// TwinCAT 3 PLC project STN100
// ProgramVersion: 3.1.4022.3
// libraries:
//   Tc2_Standard, * (Beckhoff Automation GmbH)
//   Tc2_System, * (Beckhoff Automation GmbH)
//   Tc3_Module, * (Beckhoff Automation GmbH)
// project tree:
//   ComLib/DUTs/General/ COM_ERROR_VALUE.TcTLEO, DEVICE_TYPE.TcTLEO
//   ComLib/DUTs/Level 2 Data link/ DEVICE_SEQUENCE.TcTLEO, INSTANCE_STATUS.TcTLEO
//   ComLib/DUTs/Level 4 Transport/ CommunicationData.TcDUT, DataGram.TcDUT, DATAGRAM_SEQUENCE.TcTLEO
//   ComLib/DUTs/Level 5 Session/ FUNCTION_TYPE.TcTLEO, INFO_FUNCTION_NUMBER.TcTLEO, SessionData.TcDUT, StatusInformationData.TcDUT
//   ComLib/DUTs/Level 6 Presentation/ ABB_ASYNC_FUNCTION_NUMBER.TcDUT, ABB_STATUS_OPERATING_MODE.TcTLEO, ABB_STATUS_RUNNING_MODE.TcTLEO, ABB_SYNC_FUNCTION_NUMBER.TcTLEO, GANTRY_ASYNC_FUNCTION_NUMBER.TcTLEO, GANTRY_STATUS.TcTLEO, PositionType.TcTLEO, StationType.TcTLEO
//   ComLib/GVL/ ComGVL.TcGVL
//   ComLib/POUs/Private/ _AllocateInstance.TcPOU, _CheckInstance.TcPOU, _DataGramSize.TcPOU, _FreeInstance.TcPOU, _GetInstance.TcPOU, _GetStatusInformation.TcPOU, _SetInstance.TcPOU, _TryOut.TcPOU (excluded from build)
//   ComLib/POUs/Public/Level 1 Physical/ NodeGetStatus.TcPOU, NodeGetType.TcPOU, NodeReadStrobe.TcPOU, NodeReadWord.TcPOU, NodeWriteStrobe.TcPOU, NodeWriteWord.TcPOU, ToAddress.TcPOU
//   ComLib/POUs/Public/Level 2 Data link/ DeviceCancel.TcPOU, DeviceClose.TcPOU, DeviceOpen.TcPOU, DeviceRead.TcPOU, DeviceStatus.TcPOU, DeviceUse.TcPOU, DeviceWrite.TcPOU
//   ComLib/POUs/Public/Level 4 Transport/ Communicator.TcPOU, DatagramCheckSum.TcPOU
//   ComLib/POUs/Public/Level 5 Session/RPC Remote Procedural Call/ ASyncProgress.TcPOU, ASyncRPC.TcPOU, RPC1.TcPOU, RPC2.TcPOU
//   ComLib/POUs/Public/Level 5 Session/Session/ SessionEnd.TcPOU, SessionInit.TcPOU, SessionSend.TcPOU
//   ComLib/POUs/Public/Level 6 Presentation/ABB/ ABBGetStatus.TcPOU
//   ComLib/POUs/Public/Level 6 Presentation/ABB/Goto/ ABBGoToConveyor1.TcPOU, ABBGoToConveyor2.TcPOU, ABBGoToHome.TcPOU, ABBGoToSensor.TcPOU, ABBGoToStorage.TcPOU, ABBGoToTable.TcPOU
//   ComLib/POUs/Public/Level 6 Presentation/ABB/IO/ ABBIORead.TcPOU, ABBIOReadValve.TcPOU, ABBIOWrite.TcPOU, ABBIOWriteValve.TcPOU
//   ComLib/POUs/Public/Level 6 Presentation/ABB/Move/ ABBMoveJAbs.TcPOU, ABBMoveJRel.TcPOU, ABBMoveLAbs.TcPOU, ABBMoveLRel.TcPOU
//   ComLib/POUs/Public/Level 6 Presentation/ABB/Pick Leave/ ABBPickLeaveConveyor1.TcPOU, ABBPickLeaveConveyor2.TcPOU, ABBPickLeaveSensor.TcPOU, ABBPickLeaveStorage.TcPOU, ABBPickLeaveTable.TcPOU, ABBProcessAssembly.TcPOU
//   ComLib/POUs/Public/Level 6 Presentation/Gantry/ GantryLeave.TcPOU, GantryPick.TcPOU, GantryStatus.TcPOU
//   ComLib/POUs/Public/Level 6 Presentation/ GetStatus.TcPOU
//   ComLib/VISUs/Object/ _VisuABBGoTo.TcVIS, _VisuABBPickLeave.TcVIS, _VisuABBStatus.TcVIS, _VisuAddressSelector.TcVIS, _VisuAddressShow.TcVIS, _VisuCommunicator.TcVIS, _VisuFunctionCall.TcVIS, _VisuGantryPickLeave.TcVIS, _VisuRPCStatusShow.TcVIS
//   ComLib/VISUs/ _TryOut.TcVIS (excluded from build)
//   / GlobalTextList.TcGTLO, PlcTask.TcTTO, Visualization Manager.TcVMO (not stored), VISU_TASK.TcTTO
//   GVLs/ GVL.TcGVL
//   POUs/ MAIN.TcPOU, PLC_PRG.TcPOU
//   VISUs/ Visualization.TcVIS
// real-time tasks:
//   TASK PlcTask: cycle T#10ms, priority 20, ADS port 350
//   TASK VISU_TASK: cycle T#100000us, priority 30, ADS port 351
// I/O:
//   DEVICE Device 1 (EtherCAT), AmsNetId 5.49.18.110.2.1
//     Term 1 (EK1200) [EK1200-5000 EtherCAT Power supply (2A E-Bus)]
//       Term 2 (EL6731) [EL6731 PROFIBUS DP Master]
//       Term 3 (EK1110) [EK1110 EtherCAT extension]
//     Term 4 (EK1100) [EK1100 EtherCAT Coupler (2A E-Bus)]
//       Term 5 (EL1008) [EL1008 8Ch. Dig. Input 24V, 3ms]
//       Term 6 (EL1008) [EL1008 8Ch. Dig. Input 24V, 3ms]
//       Term 7 (EL2008) [EL2008 8Ch. Dig. Output 24V, 0.5A]
//       Term 8 (EL2008) [EL2008 8Ch. Dig. Output 24V, 0.5A]
//       Term 9 (EK1110) [EK1110 EtherCAT extension]
//   DEVICE Device 2 (EL6731), AmsNetId 5.49.18.110.3.1
//     Box 10 (GSD Box) (Anybus-CC PROFIBUS DP-V1) // Vendor: HMS Industrial Networks Revision: 1.04
// variable links:
//   STN100/STN100 Instance <-> Device 1 (EtherCAT)/Term 4 (EK1100)/Term 6 (EL1008)
//     PlcTask Inputs/GVL.ixControlStnBit1 <-> Channel 1/Input
//     PlcTask Inputs/GVL.ixControlStnBit2 <-> Channel 2/Input
//     PlcTask Inputs/GVL.ixControlStnBit4 <-> Channel 3/Input
//     PlcTask Inputs/GVL.ixControlStnBit8 <-> Channel 4/Input
//     PlcTask Inputs/GVL.ixEmergencyStopActivated <-> Channel 8/Input
//     PlcTask Inputs/GVL.ixLightBeamAndGatesClosed <-> Channel 7/Input
//   STN100/STN100 Instance <-> Device 2 (EL6731)/Box 10 (GSD Box) (Anybus-CC PROFIBUS DP-V1)
//     PlcTask Inputs/ComGVL._iwABB <-> Module 5 (Input 1 word)/Inputs/Input 1 word_0_0
//     PlcTask Outputs/ComGVL._qwABB <-> Module 6 (Output 1 words)/Outputs/Output 1 words_1_0

CONFIGURATION STN100
    RESOURCE PLC ON TwinCAT3
        TASK PlcTask(INTERVAL := T#10ms, PRIORITY := 20);
        TASK VISU_TASK(INTERVAL := T#100000us, PRIORITY := 30);
        PROGRAM MAIN WITH PlcTask : MAIN;
        PROGRAM VisuElems_Visu_Prg WITH VISU_TASK : VisuElems.Visu_Prg;
    END_RESOURCE
END_CONFIGURATION

// ---- ComLib/DUTs/General/COM_ERROR_VALUE.TcTLEO
{library public}

(* Common error values for communication blocks *)
TYPE COM_ERROR_VALUE :
(
	COM_ERR_NOT_ENABLED:=-1,						(* En signal is false or block is not enabled *)
	COM_ERR_NO_ERROR:=0,							(* No error *)

 	(* Level 1 Errors *)
	COM_ERR_LEVEL1,									(* The physical layer failed during communication *)
	COM_ERR_LEVEL1_TIME_OUT,						(* Time out in the physical layer *)

 	(* Level 2 Errors *)
	COM_ERR_NOT_ALLOCATED,							(* Instance not allocated *)
	COM_ERR_INSTANCE,								(* Instance address (station/device) number not set or wrong *)
	COM_ERR_LEVEL2_TIME_OUT,						(* Time out in communication with device *)
	COM_ERR_LEVEL2_ERROR,							(* Error during send/receive *)
	COM_ERR_CANCEL,									(* Current operation was cancelled *)

 	(* Level 3 Errors *)
	COM_ERR_TWO_INSTANCES_OF_COMMUNICATOR,			(* Two instances of the communicator block exist in the configuration remove one *)
	COM_ERR_CHECKSUM,								(* Checksum error during datagram transfer *)

	(* Level 5 Error *)
	COM_ERR_NO_VALID_FUNCTION						(* Calls to an unknown RPC function *)
);
END_TYPE
//  COM_ERR_NOT_ENABLED = '-1'

// ---- ComLib/DUTs/General/DEVICE_TYPE.TcTLEO
{library PUBLIC}
TYPE DEVICE_TYPE :
(
	TYPE_ERROR:=-1, TYPE_SIMULATED:=0,  TYPE_ABB_1:=1, TYPE_GANTRY_1:=2
);
END_TYPE
//  TYPE_ERROR = '-1'

// ---- ComLib/DUTs/Level 2 Data link/DEVICE_SEQUENCE.TcTLEO
{library PUBLIC}
(*
Sequence for a specific device during send or receive on level 2.
This can be used for debug but is only visible inside a block.
 *)
TYPE DEVICE_SEQUENCE :
(
	DEVICE_SEQUENCE_NOP:=0,							(* No operation - free *)
	DEVICE_SEQUENCE_INIT,							(* Init of block *)
	DEVICE_SEQUENCE_WAIT_FOR_DEVICE_READY,			(* Prepare for wait and set busy to true *)
	DEVICE_SEQUENCE_WAIT_FOR_STROBE_LOW,			(* Wait until target device strobe and data are 0 *)
	DEVICE_SEQUENCE_PREPARE_SEND_RECEIVE,
	DEVICE_SEQUENCE_STROBE_HIGH,
	DEVICE_SEQUENCE_SEND_RECEIVE,					(* Transfer or read data *)
	DEVICE_SEQUENCE_ACK,
	DEVICE_SEQUENCE_WAIT_FOR_ANSWER,
	DEVICE_SEQUENCE_SET_LOW,						(* Data and strobe to 0 *)
	DEVICE_SEQUENCE_READY,							(* End of sequence will wait in this step until En=false *)

	DEVICE_SEQUENCE_TIME_OUT:=-1,					(* Tinme out during send or receive *)
	DEVICE_SEQUENCE_CANCEL:=-2,						(* An ongoing operation was canceld *)
	DEVICE_SEQUENCE_ERROR:=-3						(* An error during send/receive *)
);
END_TYPE
//  DEVICE_SEQUENCE_TIME_OUT = '-1'
//  DEVICE_SEQUENCE_CANCEL = '-2'
//  DEVICE_SEQUENCE_ERROR = '-3'

// ---- ComLib/DUTs/Level 2 Data link/INSTANCE_STATUS.TcTLEO
{library PUBLIC}
(*
 Status word for a specific device instance .
Function block DeviceUse or DeviceStatus will give you the status for a specific instance.
*)
TYPE INSTANCE_STATUS  : 
(
 	INSTANCE_STATUS_FREE:=0,							(* Instance not allocated *)
 	INSTANCE_STATUS_READY :=1,							(* Instance ready *)
 	INSTANCE_STATUS_BUSY:=2,							(* Instance is busy *)
	INSTANCE_STATUS_UNKNOWN:=3,							(* Unknown or address error *)

 	INSTANCE_STATUS_CANCEL:=-1							(* Instance cancel operation *)
);
END_TYPE
//  INSTANCE_STATUS_CANCEL = '-1'

// ---- ComLib/DUTs/Level 4 Transport/CommunicationData.TcDUT
{library PUBLIC}
(*
This is the data handler for all communications blocks.
Do not change any values inside the structure instead use existing function blocks to manipulate the data.
*)
TYPE CommunicationData :
STRUCT
	_Instance: 				BOOL := FALSE;								(*To check that we only have one instance of the communicator function block only one Instance can be true *)
	_ErrorID:				COM_ERROR_VALUE := COM_ERROR_VALUE.COM_ERR_NO_ERROR;			(* Current error value *)
	_Error:					BOOL:=FALSE	;								(* True if any error *)
	_Address:				INT:=-1;									(* Address value for device *)

	_Session:				SessionData;								(* Session data *)

	_ASyncProgress:			INT:=0;										(* Asynchronous function progress *)
	_ASyncStatus:			StatusInformationData;						(* Asynchronous function call status *)
	_ASyncStatusCounter:	UDINT:=0;									(* Counter to keep track of number of status calls *)

	_DataCounter:			UDINT:=0;									(* Datagram bytes transfered counter *)
	_DataExecute:			UDINT:=0;									(* Current datagram BYTE counter (EQ TO _DatatCounter OR <_DataCounter+SIZEOF DataGram) *)
	_Data:					DataGram;									(* Current datagram values*)
	_DataAnswer:			DataGram;									(* Datagram answer  *)

	_Status:				DATAGRAM_SEQUENCE := DATAGRAM_SEQUENCE.DATAGRAM_SEQUENCE_NOP;	(* Current status *)

	_TimeOutDevice:			TIME:=ComGvl.DEVICE_DEFAULT_TIME_OUT;				(* Device time out time *)
END_STRUCT
END_TYPE

// ---- ComLib/DUTs/Level 4 Transport/DataGram.TcDUT
{library PUBLIC}
(*
Structure to handle datagrams on level 4.
*)
TYPE DataGram :
STRUCT
	ParameterDW:		DWORD;		(* Parameter value (32 bit), purpose dependent on type of function *)
	ParameterB:			BYTE;		(* Parameter value (8 bit), purpose dependent on type of function *)

	FunctionType:		BYTE;		(* Type of function (8 bit) specifies a set of functions, the number must be based on the enumeration FUNCTION_TYPE, note that an enumeration is 16 bit and must be converted with WORD_TO_BYTE() to fit in this structure *)
	FunctionNumber: 	BYTE;		(* Specific Function (8 bit) *)

	CheckSum:			BYTE;		(* Checksum for DataGram *)
END_STRUCT
END_TYPE

// ---- ComLib/DUTs/Level 4 Transport/DATAGRAM_SEQUENCE.TcTLEO
{library PUBLIC}

(* Sequence for a specific communicator during send or receive *)
TYPE DATAGRAM_SEQUENCE : (
	DATAGRAM_SEQUENCE_ERROR:=-1,
	DATAGRAM_SEQUENCE_INIT:=-0,
	DATAGRAM_SEQUENCE_NOP,							(* No operation - free *)
	DATAGRAM_SEQUENCE_INIT_SEND,
	DATAGRAM_SEQUENCE_SEND_1,
	DATAGRAM_SEQUENCE_SEND_2,
	DATAGRAM_SEQUENCE_SEND_3,

	DATAGRAM_SEQUENCE_INIT_RECEIVE,
	DATAGRAM_SEQUENCE_RECEIVE_1,
	DATAGRAM_SEQUENCE_RECEIVE_2,
	DATAGRAM_SEQUENCE_RECEIVE_3,

	DATAGRAM_SEQUENCE_DONE
);
END_TYPE
//  DATAGRAM_SEQUENCE_ERROR = '-1'
//  DATAGRAM_SEQUENCE_INIT = '-0'

// ---- ComLib/DUTs/Level 5 Session/FUNCTION_TYPE.TcTLEO
{library PUBLIC}
(*
 Function type, to be used in DataGram structure to specify set of functions.

 Note that values <=0 are return values only.
 *)
TYPE FUNCTION_TYPE : 
(
	FUNCTION_TYPE_ERROR_BUSY:=-2,				(* Old function call is not ready  *)
	FUNCTION_TYPE_ERROR_NO_FUNCTION:=-1,		(* RPC function not found *)
	FUNCTION_TYPE_TASK_STARTED:=0,				(* ASynchronous function started *)
	FUNCTION_TYPE_ASYNC_RPC:=1,					(* ASynchronous RPC *)
	FUNCTION_TYPE_SYNC_RPC,   					(* Synchronous RPC *)
	FUNCTION_TYPE_INFORMATION					(* Synchronous RPC dedicated for status functions *)
);
END_TYPE
//  FUNCTION_TYPE_ERROR_BUSY = '-2'
//  FUNCTION_TYPE_ERROR_NO_FUNCTION = '-1'

// ---- ComLib/DUTs/Level 5 Session/INFO_FUNCTION_NUMBER.TcTLEO
{library PUBLIC}
TYPE INFO_FUNCTION_NUMBER :(
	INFO_FUNCTION_RPC_STATUS:=1,				(* Get RPC call status *)
	INFO_FUNCTION_SYSTEM_STATUS:=2				(* Get system status *)
);
END_TYPE

// ---- ComLib/DUTs/Level 5 Session/SessionData.TcDUT
{library PRIVATE}
(*
This is the session handler for all session blocks.
This structure can not be used outside of the CommunicationStructure.
Do not change any values inside the structure instead use existing function blocks to manipulate the data.
*)

TYPE SessionData :
STRUCT
	_Locked:			BOOL:=FALSE;				(* A session lock for this struct *)
	_SessionBussy:		BOOL:=FALSE;				(* If session is bussy sending data *)
	_SessionID:			INT:=0;						(* Session ID that locked this *)
	_SessionCounter:	INT:=0;						(* Sesion counter *)
END_STRUCT
END_TYPE

// ---- ComLib/DUTs/Level 5 Session/StatusInformationData.TcDUT
{library PUBLIC}
TYPE StatusInformationData :
STRUCT
	Progress:			INT:=0;					(* Progress on current RPC call 0-100 *)
	FunctionNumber:		INT:=0;					(* Curent RPC function number *)
	ReturnValue:		INT:=0;					(* Return value from previous RPC call *)
	Extra:				INT:=0;					(* Extra information *)
END_STRUCT
END_TYPE

// ---- ComLib/DUTs/Level 6 Presentation/ABB_ASYNC_FUNCTION_NUMBER.TcDUT
{library PUBLIC}
TYPE ABB_ASYNC_FUNCTION_NUMBER :(

	(* GoTo functions - No parameters *)
	ABB_ASYNC_FUNCTION_GOTO_HOME:=			11,
	ABB_ASYNC_FUNCTION_GOTO_TABLE:=			12,
	ABB_ASYNC_FUNCTION_GOTO_SENSOR:=		13,
	ABB_ASYNC_FUNCTION_GOTO_STORAGE:=		14,
	ABB_ASYNC_FUNCTION_GOTO_CONVEYOR_1:=	15,
	ABB_ASYNC_FUNCTION_GOTO_CONVEYOR_2:=	16,

	(* Pick Leav functions
	ParameterB=1 (TRUE) pick, 0 (FALSE) leave,
	ParameterW=position (if several positions exist)
	Note that Gripper is not affected by ParameterB value use separate function open or close gripper
 	*)
	ABB_ASYNC_FUNCTION_PL_TABLE:=			22,			(* Position 1=brick, 2=Rod, 3=Assembly *)
	ABB_ASYNC_FUNCTION_PL_SENSOR:=			23,
	ABB_ASYNC_FUNCTION_PL_STORAGE:=			24,  		(* Position 1-9 *)
	ABB_ASYNC_FUNCTION_PL_CONVEYOR_1:=		25,
	ABB_ASYNC_FUNCTION_PL_CONVEYOR_2:=		26,

	(* Process functions - No parameters *)
	ABB_ASYNC_FUNCTION_PROCESS_ASSEMBLY:=	32,

	(* Move functions
	Note, that xyz, rx,ry and rz must first be set by call to set functions (SYNC) *)
	ABB_ASYNC_ABS_MOVEJ_TO_POSE:=			101,
	ABB_ASYNC_ABS_MOVEL_TO_POSE:=			102,

	ABB_ASYNC_REL_MOVEJ_TO_POSE:=			111,
	ABB_ASYNC_REL_MOVEL_TO_POSE:=			112
);
END_TYPE

// ---- ComLib/DUTs/Level 6 Presentation/ABB_STATUS_OPERATING_MODE.TcTLEO
{library PUBLIC}
TYPE ABB_STATUS_OPERATING_MODE :
(
	ABB_STATUS_OPERATION_UNDEF:=0,				(* Undefined operating mode *)
	ABB_STATUS_OPERATION_AUTO:=1,				(* Automatic operating mode *)
	ABB_STATUS_OPERATION_MAN_PROG:=2, 			(* Manual operating mode MAX. 250 mm/S *)
	ABB_STATUS_OPERATION_MAN_TEST:=3 			(* Manual operating mode full speed, 100 % *)
);
END_TYPE

// ---- ComLib/DUTs/Level 6 Presentation/ABB_STATUS_RUNNING_MODE.TcTLEO

TYPE ABB_STATUS_RUNNING_MODE :
(
	ABB_STATUS_RUN_UNDEF:=0, 			(* Undefined running mode *)
	ABB_STATUS_RUN_CONT_CYCLE:=1, 		(* Continuous or cycle running mode *)
	ABB_STATUS_RUN_INSTR_FWD:=2,		(* Instruction forward running mode *)
	ABB_STATUS_RUN_INSTR_BWD:=3, 		(* Instruction backward running mode *)
	ABB_STATUS_RUN_SIM:=4, 				(* Simulated running mode *)
	ABB_STATUS_RUN_STEP_MOVE:=5 		(* MOVE instructions in forward running mode and logical instructions in continuous running mode *)
);
END_TYPE

// ---- ComLib/DUTs/Level 6 Presentation/ABB_SYNC_FUNCTION_NUMBER.TcTLEO
{library PUBLIC}
TYPE ABB_SYNC_FUNCTION_NUMBER :(
(* Set variable values
	ParameterW is the new value *)
	ABB_SYNC_FUNCTION_SET_X:=11,
	ABB_SYNC_FUNCTION_SET_Y:=12,
	ABB_SYNC_FUNCTION_SET_Z:=13,
	ABB_SYNC_FUNCTION_SET_RX:=14,
	ABB_SYNC_FUNCTION_SET_RY:=15,
	ABB_SYNC_FUNCTION_SET_RZ:=16,

(* Get variable values *)
	ABB_SYNC_FUNCTION_GET_X:=21,
	ABB_SYNC_FUNCTION_GET_Y:=22,
	ABB_SYNC_FUNCTION_GET_Z:=23,
	ABB_SYNC_FUNCTION_GET_RX:=24,
	ABB_SYNC_FUNCTION_GET_RY:=25,
	ABB_SYNC_FUNCTION_GET_RZ:=26,

(* Set pneumatic valve value
	ParameterB=1 or 0 *)
	ABB_SYNC_SET_VALVE1:=31,
	ABB_SYNC_SET_VALVE2:=32,
	ABB_SYNC_SET_VALVE3:=33,

	ABB_SYNC_GET_VALVE1:=41,
	ABB_SYNC_GET_VALVE2:=42,
	ABB_SYNC_GET_VALVE3:=43,

	ABB_SYNC_READ_DI:=101,
	ABB_SYNC_WRITE_DO:=102

);
END_TYPE

// ---- ComLib/DUTs/Level 6 Presentation/GANTRY_ASYNC_FUNCTION_NUMBER.TcTLEO
{library PUBLIC}
TYPE GANTRY_ASYNC_FUNCTION_NUMBER :(

(* GoTo functions - No parameters *)
	GANTRY_ASYNC_FUNCTION_GOTO_HOME:=		11,
	GANTRY_ASYNC_FUNCTION_GOTO_STATION:=	12,

(* Pick Leav function
	ParameterW=Station 1-4*10 + position 1-9 + Station 1-4*1000 +position 1-9 * 100
 *)
	GANTRY_ASYNC_FUNCTION_PL:=					22			(* Pick/leave at position *)
);
END_TYPE

// ---- ComLib/DUTs/Level 6 Presentation/GANTRY_STATUS.TcTLEO
{library PUBLIC}
TYPE GANTRY_STATUS :
(
	GANTRY_STATUS_NOT_ENABLED:=-1,					(* En signal is false or block is not enabled *)
	GANTRY_STATUS_NOT_READY:=0,						(* NOT ready *)
	GANTRY_STATUS_READY:=1, 							(* Auto run OK *)
	GANTRY_STATUS_INIT_MOVE:=2, 						(* Init of accelerations speeds etc *)
	GANTRY_STATUS_START_MOVE:=3,					(* Start transportation *)
	GANTRY_STATUS_MOVE_TO_STATION:=4,				(* Robot in motion *)
	GANTRY_STATUS_WAIT_CLEAR_ORDER:=5,			(* Wait until order is cleared *)
	GANTRY_STATUS_WAIT_FOR_ORDER:=6,				(* Wait for a pick or leave order *)
	GANTRY_STATUS_ORDER_ERROR:=7,				(* Error in pick or leave order *)
	GANTRY_STATUS_MOVE_TO_PICK:=8,					(* Robot picks pallet *)
	GANTRY_STATUS_WAIT_FOR_LEAVE_ORDER:=9,	(* Wait for leave order *)
	GANTRY_STATUS_ORDER_LEAVE_ERROR:=10,		(* Error in leave order *)
	GANTRY_STATUS_MOVE_TO_LEAVE:=11 				(* Robot leave pallet *)
);
END_TYPE
//  GANTRY_STATUS_NOT_ENABLED = '-1'

// ---- ComLib/DUTs/Level 6 Presentation/PositionType.TcTLEO
{library PUBLIC}
(* Position number type *)
TYPE PositionType : INT(1..9);
END_TYPE

// ---- ComLib/DUTs/Level 6 Presentation/StationType.TcTLEO
{library PUBLIC}
(* Station number type *)
TYPE StationType : INT(1..9);
END_TYPE

// ---- ComLib/GVL/ComGVL.TcGVL
{attribute 'qualified_only'}
{library PUBLIC}
VAR_GLOBAL CONSTANT
	VERSION_COM_LIBRARY:					REAL:=3.0;		(* Version number for library *)
	DEVICE_DEFAULT_TIME_OUT:		 		TIME := T#1S;	(* Default time out for single word messages to a specific device *)
END_VAR

{library private}
VAR_GLOBAL CONSTANT
	INSTANCE_MAX_NUMBER_OF_STATIONS:		INT := 6;
	INSTANCE_MAX_NUMBER_OF_DEVICES:			INT := 2;

	ADDRESS_SIMULATED:						INT := 602;
END_VAR

{library private}
VAR_GLOBAL
	
	//ProfiBusDP Communication to ABB-robot or Portal Robot (Gantry)
	{attribute 'TcSwapWord'}
	_iwABB     AT %I* : WORD;	//From ABB robot (Swaped byte order)
	_iw1Gantry AT %I* : WORD;	//From Gantry robot
	_iw2Gantry AT %I* : WORD;	
	_iw3Gantry AT %I* : WORD;	

	{attribute 'TcSwapWord'}
	_qwABB 	   AT %Q* : WORD; //To ABB robot (Swaped Byte order)
	_qw1Gantry AT %Q* : WORD; //To Gantry robot 
	_qw2Gantry AT %Q* : WORD; //To Gantry robot 
	_qw3Gantry AT %Q* : WORD; //To Gantry robot 
	
	
	




	_Instance : ARRAY  [1..INSTANCE_MAX_NUMBER_OF_STATIONS,
						   1..INSTANCE_MAX_NUMBER_OF_DEVICES]
													OF  INSTANCE_STATUS;

(*	Index 1: 1=PLC, 2="Simulated Robot",
	Index 2: 1=Strobe, 2=data  *)	
	_DataSimulatedStation:	ARRAY [1..INSTANCE_MAX_NUMBER_OF_DEVICES, 1..2] OF BYTE;


(*|                         |                                     | *)
(*|                         |                                     | *)
(*V                         V                                     V *)
(* -----------------------------------------------------------------*)


(*

(* Global Try Out variables only used by the TryOut block *)

(* Try out Communicator *)
	_miAddressNumber:			ARRAY [1..5] OF INT := [101, 201, 301, 401, 502];
	_miAddressIndex:			INT:=1;
	_fbTryOutCommunicator:		Communicator;
	_msTryOutData: 				CommunicationData;
	_mxTryOutEnable:			BOOL;

	_glAddressNameTable: 		ARRAY [1..5] OF STRING:= ['Station 100' , 'Station 200', 'Station 300', 'Station 400',  'Station 500'];
	_glAddressSelectionIndex: 	INT:=1;

	_glErrorTable:				ARRAY [ -1 .. 10] OF STRING :=
	 	['En signal is false or block is not enabled',
		 'No error',
		 'The physical layer failed during communication',
		 'Time out in the physical layer',
		 'Instance not allocated',
		 'Instance address (station/device) number not set or wrong',
		 'Time out in communication with device',
		 'Error during send/receive',
		 'Current operation was cancelled',
		 'Two instances of the communicator block exist in the configuration remove one',
		 'Checksum error during datagram transfer',
		 'Calls to an unknown RPC function'];

	_fbTryOutGetStatus:					GetStatus;
	_fbTryOutGetStatusRunning:			BOOL;
	_fbTryOutGetStatusProgress:			INT;
	_fbTryOutGetStatusProgramNumber:	INT;
	_fbTryOutGetStatusHeartBeat:		BOOL;
	_fbTryOutGetStatusError: 			BOOL;

(* ABB Functions *)
	_fbTryOutShowABB:					BOOL;

	_fbTryOutDone:						BOOL;
	_fbTryOutExecuting:					BOOL;
	_fbTryOutWaiting:					BOOL;
	_fbTryOutError:						BOOL;
	_fbTryOutProgress:					INT;

	_fbTryOutABBGetStatus:				ABBGetStatus;
	_fbTryOutABBRunMode:				ABB_STATUS_RUNNING_MODE;
	_fbTryOutABBOpMode:					ABB_STATUS_OPERATING_MODE;

	_gABBRunTable:						ARRAY [1 .. 6] OF STRING :=
		['Undefined running mode',
		'Continuous or cycle running mode',
		'Instruction forward running mode',
		'Instruction backward running mode',
		'Simulated running mode',
		'MOVE instr. in forward running and logical instr. in continuous running mode'];

	_gABBOpTable:						ARRAY [ 1 .. 4] OF STRING :=
		['Undefined operating mode',
		'Automatic operating mode',
		'Manual operating mode MAX. 250 mm/S',
		'Manual operating mode full speed, 100 %'];

	_fbTryOutABBGoToHome:				ABBGoToHome;
	_fbTryOutABBGoToHomeEn:				BOOL;

	_fbTryOutABBGoToSensor:				ABBGoToSensor;
	_fbTryOutABBGoToSensorEn:			BOOL;

	_fbTryOutABBGoToStorage:			ABBGoToStorage;
	_fbTryOutABBGoToStorageEn:			BOOL;

	_fbTryOutABBGoToTable:				ABBGoToTable;
	_fbTryOutABBGoToTableEn:			BOOL;

	_fbTryOutABBGoToConveyor1:			ABBGoToConveyor1;
	_fbTryOutABBGoToConveyor1En:		BOOL;

	_fbTryOutABBGoToConveyor2:			ABBGoToConveyor2;
	_fbTryOutABBGoToConveyor2En:		BOOL;

	_fbTryOutABBPickLeaveSensor:		ABBPickLeaveSensor;
	_fbTryOutABBPickLeaveSensorEn:		BOOL;
	_fbTryOutABBPSensor:				BOOL;

	_fbTryOutABBPickLeaveStorage:		ABBPickLeaveStorage;
	_fbTryOutABBPickLeaveStorageEn:		BOOL;
	_fbTryOutABBPStorage:				BOOL;
	_fbTryOutABBPStoragePos:			INT:=1;

	_fbTryOutABBPickLeaveTable:			ABBPickLeaveTable;
	_fbTryOutABBPickLeaveTableEn:		BOOL;
	_fbTryOutABBPTable:					BOOL;
	_fbTryOutABBPTablePos:				INT:=1;

	_fbTryOutABBPickLeaveConveyor1:		ABBPickLeaveConveyor1;
	_fbTryOutABBPickLeaveConveyor1En:	BOOL;
	_fbTryOutABBPConveyor1:				BOOL;

	_fbTryOutABBPickLeaveConveyor2:		ABBPickLeaveConveyor2;
	_fbTryOutABBPickLeaveConveyor2En:	BOOL;
	_fbTryOutABBPConveyor2:				BOOL;

(* Gantry Functions *)
	_fbTryOutShowGantry:			BOOL;

	_fbTryOutGantryPick:			GantryPick;
	_fbTryOutGantryPickEn:			BOOL;
	_fbTryOutGantryPickStation:		INT:=1;
	_fbTryOutGantryPickPos:			INT:=1;

	_fbTryOutGantryLeave:			GantryLeave;
	_fbTryOutGantryLeaveEn:			BOOL;
	_fbTryOutGantryLeaveStation:	INT:=1;
	_fbTryOutGantryLeavePos:		INT:=2;
*)
END_VAR

// ---- GVLs/GVL.TcGVL
{attribute 'qualified_only'}
VAR_GLOBAL
	

	//OPC-UA Communication to STN500 (the crane)
	{attribute 'OPC.UA.DA' := '1'}
	iToSTN500FromSTN100 : ARRAY[1..8] OF INT; (* To STN500 *)

	{attribute 'OPC.UA.DA' := '1'}
	iFromSTN500ToSTN100 : ARRAY[1..8] OF INT; (* From STN500 *)

	
	//Inputs from the sensors in controlstation
	ixControlStnBit1 AT %I* : BOOL;	
	ixControlStnBit2 AT %I* : BOOL;
	ixControlStnBit4 AT %I* : BOOL;
	ixControlStnBit8 AT %I* : BOOL;
	
	

	
	(* Gates and emergency stop, status signal *)
	ixLightBeamAndGatesClosed 	AT %I* : BOOL;
	ixEmergencyStopActivated 	AT %I* : BOOL;
	
	
	(* Light staple *)
	qxLampRed 		AT %Q*: BOOL;
	qxLampYellow 	AT %Q*: BOOL;
	qxLampGreen 	AT %Q*: BOOL;
	
	
	
END_VAR

// ---- POUs/MAIN.TcPOU
PROGRAM MAIN
VAR

END_VAR

PLC_PRG();

END_PROGRAM

// ---- POUs/PLC_PRG.TcPOU
PROGRAM PLC_PRG
VAR
	//Visualisation buttons	
	mxButtonReset	: BOOL;	
	mxButtonStart: BOOL;

	//Internal use
	mxStart: BOOL;
	mxDone: BOOL;
	mxComBusy: BOOL;
	CommData: CommunicationData;	
	
	//Motion Function Blocks
	fbCommunicator: Communicator;
	fbABBGoToHome_1: ABBGoToHome;
	fbABBGoToTable_1: ABBGoToTable;
END_VAR

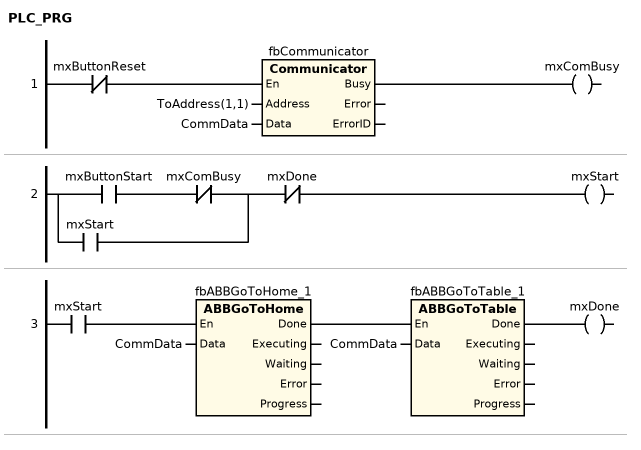
// NETWORK 1
fbCommunicator(En := NOT mxButtonReset, Address := ToAddress(1,1), Data := CommData); // Communicator
mxComBusy := fbCommunicator.Busy;

// NETWORK 2
mxStart := (mxButtonStart AND NOT mxComBusy OR mxStart) AND NOT mxDone;

// NETWORK 3
fbABBGoToHome_1(En := mxStart, Data := CommData); // ABBGoToHome
fbABBGoToTable_1(En := fbABBGoToHome_1.Done, Data := CommData); // ABBGoToTable
mxDone := fbABBGoToTable_1.Done;

END_PROGRAM

// ---- ComLib/POUs/Public/Level 4 Transport/Communicator.TcPOU
{library PUBLIC}
(* Communication interface on level 4 to be used as a single access point to communicate with external equipment (device).
    Note, that you must make one and only one instance per address (device) of this block. This block instance 
    coordinates all communication actions from all POUs to a specific device.

   The Data input must be connected to a common variable of the type CommunicationData. 
   The Data variable must then be used together with all function blocks that want to communicate with
   the specified equipment. It is possible to use function blocks on level 4-6 together with the communicator.
  However, note that it is not possible to utilize function blocks on level 1-3 together with the communicator.
*)
FUNCTION_BLOCK Communicator
VAR_INPUT
	En: 				BOOL:=TRUE;						(* Enable signal must be true during communication, set to false (pulse) to reset error and restart the block.  *)
	Address :			INT:=-1;						(* Address is the station number + device number, e.g.  202, 301, 404 and must be constant during run you can use ToAddress() function to calculate an address. *)
END_VAR
VAR_OUTPUT
	Busy: 				BOOL:=FALSE;					(* Busy is true if the block is communicating with target, otherwise false. *)
	Error: 				BOOL:=FALSE;					(* True if any error, to reset error set En to low and then back to high*)
	ErrorID: 			COM_ERROR_VALUE:=COM_ERROR_VALUE.COM_ERR_NO_ERROR;	(* The error number, if no error the output is equal to COM_ERR_NO_ERROR i.e., 0 *)
END_VAR
VAR_IN_OUT
	Data:				 CommunicationData;				(* Common data structure to connect all communication blocks that want to access this block *)
END_VAR
{library private}
VAR
	AllowToRun:		BOOL:=FALSE	;						(* If we are alone then we are allow to execute the communication*)
	Instance:		INT:=-1;							(* Device instance number *)
	DeviceType:		DEVICE_TYPE:=DEVICE_TYPE.TYPE_ERROR;
	InstanceStatus: INSTANCE_STATUS;
	Sequence: 		DATAGRAM_SEQUENCE:=DATAGRAM_SEQUENCE.DATAGRAM_SEQUENCE_INIT;
	ENWrite: 		BOOL:=FALSE;
	ENRead: 		BOOL:=FALSE;

	DataPointer:	POINTER TO BYTE;
	DataWord: 		WORD;
	StationNumber:	WORD;
	PositionNumber:	WORD;

	fbDeviceWrite: 	DeviceWrite;
	fbDeviceRead: 	DeviceRead;
	fbDeviceCancel: DeviceCancel;

	fbTON_TimeOut:	TON;							(* Only used for special sequence of gantry *)
	DEVICE_DEFAULT_TIME_OUT: INT;

	(* Variables used to change byte order in Data.ParameterDW *)
	DataHi1: BYTE; //Answer from ABB robot
	DataLo1: BYTE;
	DataHi2: BYTE;
	DataLo2: BYTE;
	DataSLo1: BYTE; //Send to ABB robot
	DataSHi1: BYTE;
	DataSHi2: BYTE;
	DataSLo2: BYTE;
END_VAR

IF NOT AllowToRun AND Instance=-1 AND En THEN
	InstanceStatus:=_GetInstance(Address);
	Instance:=0;
	Data._Address:=Address;

	IF InstanceStatus=INSTANCE_STATUS.INSTANCE_STATUS_FREE THEN
		IF DeviceOpen(Address) THEN
			Instance:=Address;
			DeviceType:=NodeGetType(Address);
			AllowToRun:=TRUE;
			Data._Instance:=TRUE;
			Error:=FALSE;
			ErrorID:=COM_ERROR_VALUE.COM_ERR_NO_ERROR;
		END_IF;
	ELSE
		Error:=TRUE;
		CASE InstanceStatus OF
			INSTANCE_STATUS.INSTANCE_STATUS_READY,  INSTANCE_STATUS.INSTANCE_STATUS_BUSY,  INSTANCE_STATUS.INSTANCE_STATUS_CANCEL:
					ErrorID:=COM_ERROR_VALUE.COM_ERR_TWO_INSTANCES_OF_COMMUNICATOR;

			INSTANCE_STATUS.INSTANCE_STATUS_UNKNOWN:
				ErrorID:=COM_ERROR_VALUE.COM_ERR_INSTANCE;
		END_CASE;
	END_IF;
END_IF;

IF AllowToRun THEN
	IF Address<>Data._Address THEN
		Busy:=FALSE;
		Error:=TRUE;
		ErrorID:=COM_ERROR_VALUE.COM_ERR_INSTANCE;
		RETURN;
	END_IF;

	fbDeviceWrite(En:=ENWrite AND En, Instance:=Instance, Data:=DataWord, TimeOut:=Data._TimeOutDevice);
	fbDeviceRead(En:=ENRead AND En, Instance:=Instance, TimeOut:=Data._TimeOutDevice);

	IF fbDeviceWrite.Error AND fbDeviceWrite.ErrorID<>COM_ERROR_VALUE.COM_ERR_CANCEL THEN
		Sequence:=DATAGRAM_SEQUENCE.DATAGRAM_SEQUENCE_ERROR;
		Error:=TRUE;
		ErrorID:=fbDeviceWrite.ErrorID;
	END_IF;

	IF fbDeviceRead.Error AND fbDeviceRead.ErrorID<>COM_ERROR_VALUE.COM_ERR_CANCEL THEN
		Sequence:=DATAGRAM_SEQUENCE.DATAGRAM_SEQUENCE_ERROR;
		Error:=TRUE;
		ErrorID:=fbDeviceRead.ErrorID;
	END_IF;

	IF En THEN
		IF DeviceType=DEVICE_TYPE.TYPE_ABB_1 THEN
			_SequenceABB_1();
		ELSIF DeviceType=DEVICE_TYPE.TYPE_GANTRY_1 THEN
			_SequenceGantry_1();
		ELSE
			Error:=TRUE;
			ErrorID:=COM_ERROR_VALUE.COM_ERR_INSTANCE;
		END_IF;
	ELSE (* En *)
		Sequence:=DATAGRAM_SEQUENCE.DATAGRAM_SEQUENCE_INIT;
		ENWrite:=FALSE;
		ENRead:=FALSE;
		Busy:=FALSE;
		Error:=FALSE;
		ErrorID:=COM_ERROR_VALUE.COM_ERR_NOT_ENABLED;

		Data._DataCounter:=0;
		Data._DataExecute:=0;
	END_IF (* En *)
END_IF;


(* Copy error to struct *)
Data._ErrorID:=ErrorID;
Data._Error:=Error;
Data._Status:=Sequence;

ACTION _SequenceABB_1:
CASE Sequence OF
			DATAGRAM_SEQUENCE.DATAGRAM_SEQUENCE_ERROR:
				Error:=TRUE;

			DATAGRAM_SEQUENCE.DATAGRAM_SEQUENCE_INIT:
				ErrorID:=COM_ERROR_VALUE.COM_ERR_NO_ERROR;
				fbDeviceCancel(En:=TRUE, Instance:=Instance);

				IF fbDeviceCancel.Done THEN
					(* Cancel set ok *)
					fbDeviceCancel(En:=FALSE, Instance:=Instance);

					(* Force DeviceWrite to execute cancel *)
					fbDeviceWrite(En:=TRUE, Instance:=Instance, Data:=DataWord, TimeOut:=Data._TimeOutDevice);
					Sequence:=DATAGRAM_SEQUENCE.DATAGRAM_SEQUENCE_NOP;
				END_IF;

			DATAGRAM_SEQUENCE.DATAGRAM_SEQUENCE_NOP:		(* Wait for order *)
				IF Data._DataCounter<>Data._DataExecute THEN
					Busy:=TRUE;
					Sequence:=DATAGRAM_SEQUENCE.DATAGRAM_SEQUENCE_INIT_SEND;
				END_IF;

			DATAGRAM_SEQUENCE.DATAGRAM_SEQUENCE_INIT_SEND:
				Data._Data.CheckSum:=DatagramCheckSum(Data._Data);
				DataPointer:= ADR(Data._Data);
				Sequence:=DATAGRAM_SEQUENCE.DATAGRAM_SEQUENCE_SEND_1;

				(* Change byte order for Intel CPU *)
				DataSLo2 := DWORD_TO_BYTE( Data._Data.ParameterDW AND 16#FF);
				DataSHi2 := DWORD_TO_BYTE( SHR(Data._Data.ParameterDW AND 16#FF00,8));
                DataSLo1 := DWORD_TO_BYTE( SHR(Data._Data.ParameterDW AND 16#FF000,16)); 
				DataSHi1 := DWORD_TO_BYTE( SHR(Data._Data.ParameterDW AND 16#FF000000,24));
				
				Data._Data.ParameterDW := BYTE_TO_DWORD( DataSHi1) OR SHL( BYTE_TO_DWORD( DataSLo1),8) OR 
                                                 SHL(BYTE_TO_DWORD( DataSHi2),16) OR SHL(BYTE_TO_DWORD( DataSLo2),24);
				
			DATAGRAM_SEQUENCE.DATAGRAM_SEQUENCE_SEND_1:
				DataWord:=BYTE_TO_WORD(DataPointer^);
				ENWrite:=TRUE;
				Sequence:=DATAGRAM_SEQUENCE.DATAGRAM_SEQUENCE_SEND_2;

			DATAGRAM_SEQUENCE.DATAGRAM_SEQUENCE_SEND_2:
				IF fbDeviceWrite.Done THEN
					ENWrite:=FALSE;
					Sequence:=DATAGRAM_SEQUENCE.DATAGRAM_SEQUENCE_SEND_3;
				END_IF;

			DATAGRAM_SEQUENCE.DATAGRAM_SEQUENCE_SEND_3:
				Data._DataCounter:=Data._DataCounter+1;
				DataPointer:=DataPointer+1;

				IF Data._DataCounter=Data._DataExecute THEN
					Sequence:=DATAGRAM_SEQUENCE.DATAGRAM_SEQUENCE_INIT_RECEIVE;
				ELSE
					Sequence:=DATAGRAM_SEQUENCE.DATAGRAM_SEQUENCE_SEND_1;
				END_IF;

			DATAGRAM_SEQUENCE.DATAGRAM_SEQUENCE_INIT_RECEIVE:
				DataPointer:= ADR(Data._DataAnswer);
				Data._DataExecute:=Data._DataExecute + INT_TO_UDINT( _DataGramSize());
				Sequence:=DATAGRAM_SEQUENCE.DATAGRAM_SEQUENCE_RECEIVE_1;

			DATAGRAM_SEQUENCE.DATAGRAM_SEQUENCE_RECEIVE_1:
				ENRead:=TRUE;
				Sequence:=DATAGRAM_SEQUENCE.DATAGRAM_SEQUENCE_RECEIVE_2;

			DATAGRAM_SEQUENCE.DATAGRAM_SEQUENCE_RECEIVE_2:
				IF fbDeviceRead.Done THEN
					ENRead:=FALSE;
					DataPointer^:=WORD_TO_BYTE(fbDeviceRead.Data);
					Sequence:=DATAGRAM_SEQUENCE.DATAGRAM_SEQUENCE_RECEIVE_3;
				END_IF;

			DATAGRAM_SEQUENCE.DATAGRAM_SEQUENCE_RECEIVE_3:
				Data._DataCounter:=Data._DataCounter+1;
				DataPointer:=DataPointer+1;

				IF Data._DataCounter=Data._DataExecute THEN
					Sequence:=DATAGRAM_SEQUENCE.DATAGRAM_SEQUENCE_DONE;
				ELSE
					Sequence:=DATAGRAM_SEQUENCE.DATAGRAM_SEQUENCE_RECEIVE_1;
				END_IF;

			DATAGRAM_SEQUENCE.DATAGRAM_SEQUENCE_DONE:
				Busy:=FALSE;

				(* Change byte order for Intel CPU *)
				DataLo1 := DWORD_TO_BYTE( Data._DataAnswer.ParameterDW AND 16#FF);
				DataHi1 := DWORD_TO_BYTE( SHR(Data._DataAnswer.ParameterDW AND 16#FF00,8));
                DataLo2 := DWORD_TO_BYTE( SHR(Data._DataAnswer.ParameterDW AND 16#FF000,16)); 
				DataHi2 := DWORD_TO_BYTE( SHR(Data._DataAnswer.ParameterDW AND 16#FF000000,24));
				
				Data._DataAnswer.ParameterDW := BYTE_TO_DWORD( DataHi1) OR SHL( BYTE_TO_DWORD( DataLo1),8) OR 
                                                SHL(BYTE_TO_DWORD( DataHi2),16) OR SHL(BYTE_TO_DWORD( DataLo2),24);
				
				IF Data._DataAnswer.CheckSum = DatagramCheckSum(Data._DataAnswer) THEN
					Data._Session._SessionCounter:=Data._Session._SessionCounter+1;
					Sequence:=DATAGRAM_SEQUENCE.DATAGRAM_SEQUENCE_NOP;
				ELSE
					ErrorID:= DINT_TO_INT( INT_TO_DINT( DATAGRAM_SEQUENCE.DATAGRAM_SEQUENCE_DONE));
					Error:=TRUE;
					Sequence:=DATAGRAM_SEQUENCE.DATAGRAM_SEQUENCE_DONE;
				END_IF;

		END_CASE;
END_ACTION

ACTION _SequenceGantry_1:
(* Note that the implementation for the Gantry does not use level 2 as intended
   it uses a mix of level 1 and 2 due to an older communication protocol in the UHS *)

		CASE Sequence OF
			DATAGRAM_SEQUENCE.DATAGRAM_SEQUENCE_ERROR:
				Error:=TRUE;
				NodeWriteWord(Address:=Instance, Channel:=0, Data:=0);									(* Write no order to pick position to crane *)
				NodeWriteWord(Address:=Instance, Channel:=1, Data:=0);									(* Write no order to pick position to crane *)

			DATAGRAM_SEQUENCE.DATAGRAM_SEQUENCE_INIT:
				ErrorID:=COM_ERROR_VALUE.COM_ERR_NO_ERROR;
				fbDeviceCancel(En:=TRUE, Instance:=Instance);

				IF fbDeviceCancel.Done THEN
					(* Cancel set ok *)
					fbDeviceCancel(En:=FALSE, Instance:=Instance);

					(* Force DeviceWrite to execute cancel *)
					fbDeviceWrite(En:=TRUE, Instance:=Instance, Data:=DataWord, TimeOut:=Data._TimeOutDevice);
					Sequence:=DATAGRAM_SEQUENCE.DATAGRAM_SEQUENCE_NOP;
				END_IF;

			DATAGRAM_SEQUENCE.DATAGRAM_SEQUENCE_NOP:		(* Wait for order *)
				IF Data._DataCounter<>Data._DataExecute THEN
					Busy:=TRUE;
					Sequence:=DATAGRAM_SEQUENCE.DATAGRAM_SEQUENCE_INIT_SEND;
				END_IF;

			DATAGRAM_SEQUENCE.DATAGRAM_SEQUENCE_INIT_SEND:
				IF Data._Data.FunctionType=FUNCTION_TYPE.FUNCTION_TYPE_INFORMATION AND Data._Data.FunctionNumber=INFO_FUNCTION_NUMBER.INFO_FUNCTION_RPC_STATUS THEN
					IF NodeReadWord(Address:=Instance, Channel:=0) =0 AND NodeReadWord(Address:=Instance, Channel:=1) =0 THEN
						Data._DataAnswer.ParameterDW:=0;
					ELSE
						Data._DataAnswer.ParameterDW:=1;
					END_IF;

					Sequence:=DATAGRAM_SEQUENCE.DATAGRAM_SEQUENCE_DONE;

				ELSIF Data._Data.FunctionType=FUNCTION_TYPE.FUNCTION_TYPE_ASYNC_RPC AND Data._Data.FunctionNumber=GANTRY_ASYNC_FUNCTION_NUMBER.GANTRY_ASYNC_FUNCTION_PL THEN
					Sequence:=DATAGRAM_SEQUENCE.DATAGRAM_SEQUENCE_SEND_1;
				ELSE
					ErrorID:=COM_ERROR_VALUE.COM_ERR_NO_VALID_FUNCTION;
					Error:=TRUE;
					Sequence:=DATAGRAM_SEQUENCE.DATAGRAM_SEQUENCE_ERROR;
				END_IF;

			DATAGRAM_SEQUENCE.DATAGRAM_SEQUENCE_SEND_1:
				(* Get pick order from Data.ParameterDW and send to gantry *)
				StationNumber:=DWORD_TO_WORD(Data._Data.ParameterDW/1000)*10;					(* 10-40 or 0*)

				IF StationNumber<>0 THEN
					PositionNumber:=DWORD_TO_WORD(Data._Data.ParameterDW/100)-StationNumber-1;	(* 0-8 *)
					PositionNumber:= ((PositionNumber/3)+1)*10 + (PositionNumber MOD 3)+1 ;				(* 11, 12, 13, 21, 22, 23, 31, 32, 33 *)

					DataWord:=Stationnumber*10+ PositionNumber;
					NodeWriteWord(Address:=Instance, Channel:=0, Data:=DataWord);							(* Write pick position to crane *)
					fbTON_TimeOut(IN:=FALSE);
					Sequence:=DATAGRAM_SEQUENCE.DATAGRAM_SEQUENCE_SEND_2;
				ELSE
					Sequence:=DATAGRAM_SEQUENCE.DATAGRAM_SEQUENCE_SEND_3;
				END_IF;

			DATAGRAM_SEQUENCE.DATAGRAM_SEQUENCE_SEND_2:
				(* Wait for ack of order *)
				fbTON_TimeOut(IN:=TRUE, PT:=ComGVL.DEVICE_DEFAULT_TIME_OUT);

				IF DataWord=NodeReadWord(Address:=Instance, Channel:=0) THEN
					Sequence:=DATAGRAM_SEQUENCE.DATAGRAM_SEQUENCE_SEND_3;
				ELSIF fbTON_TimeOut.Q THEN
					ErrorID:=COM_ERROR_VALUE.COM_ERR_LEVEL2_TIME_OUT;
					Sequence:=DATAGRAM_SEQUENCE.DATAGRAM_SEQUENCE_ERROR;
				END_IF;

			DATAGRAM_SEQUENCE.DATAGRAM_SEQUENCE_SEND_3:
				NodeWriteWord(Address:=Instance, Channel:=0, Data:=0);									(* Write no order to pick position to crane *)
				Sequence:=DATAGRAM_SEQUENCE.DATAGRAM_SEQUENCE_INIT_RECEIVE;

			DATAGRAM_SEQUENCE.DATAGRAM_SEQUENCE_INIT_RECEIVE:
				(* Get leave order from Data.ParameterDW*)
				StationNumber:=DWORD_TO_WORD(Data._Data.ParameterDW)-DWORD_TO_WORD(Data._Data.ParameterDW/100)*100;	(* 11-49 or 0*)

				IF StationNumber<>0 THEN
					PositionNumber:=StationNumber-(StationNumber/10)*10-1;									(* 0-8 *)
					PositionNumber:= ((PositionNumber/3)+1)*10 + (PositionNumber MOD 3) +1;				(* 11, 12, 13, 21, 22, 23, 31, 32, 33 *)
	
					StationNumber:=(StationNumber/10)*10;														(* 10-40 *)
					DataWord:=Stationnumber*10+ PositionNumber;
					NodeWriteWord(Address:=Instance, Channel:=1, Data:=DataWord);							(* Write leave position to crane *)
					fbTON_TimeOut(IN:=FALSE);
					Sequence:=DATAGRAM_SEQUENCE.DATAGRAM_SEQUENCE_RECEIVE_1;
				ELSE
					Sequence:=DATAGRAM_SEQUENCE.DATAGRAM_SEQUENCE_RECEIVE_2;
				END_IF;

			DATAGRAM_SEQUENCE.DATAGRAM_SEQUENCE_RECEIVE_1:
				(* Wait for ack. *)
				fbTON_TimeOut(IN:=TRUE, PT:=ComGVL.DEVICE_DEFAULT_TIME_OUT);

				IF DataWord=NodeReadWord(Address:=Instance, Channel:=1) THEN
					Sequence:=DATAGRAM_SEQUENCE.DATAGRAM_SEQUENCE_RECEIVE_2;
				ELSIF fbTON_TimeOut.Q THEN
					ErrorID:=COM_ERROR_VALUE.COM_ERR_LEVEL2_TIME_OUT;
					Sequence:=DATAGRAM_SEQUENCE.DATAGRAM_SEQUENCE_ERROR;
				END_IF;

			DATAGRAM_SEQUENCE.DATAGRAM_SEQUENCE_RECEIVE_2:
				NodeWriteWord(Address:=Instance, Channel:=1, Data:=0);									(* Write no order to leave position to crane *)
				Sequence:=DATAGRAM_SEQUENCE.DATAGRAM_SEQUENCE_RECEIVE_3;

			DATAGRAM_SEQUENCE.DATAGRAM_SEQUENCE_RECEIVE_3:
				Sequence:=DATAGRAM_SEQUENCE.DATAGRAM_SEQUENCE_DONE;

			DATAGRAM_SEQUENCE.DATAGRAM_SEQUENCE_DONE:
				Busy:=FALSE;
				Data._Session._SessionCounter:=Data._Session._SessionCounter+1;
				Data._DataCounter:=Data._DataExecute;
				Sequence:=DATAGRAM_SEQUENCE.DATAGRAM_SEQUENCE_NOP;
		END_CASE;
END_ACTION

END_FUNCTION_BLOCK

// ---- ComLib/POUs/Public/Level 2 Data link/DeviceWrite.TcPOU
{library PUBLIC}
(*
  Function to write a word to a specific device defined by Instance number.
  The Instance must be open (DeviceOpen or DeviceUse) before you can use DeviceWrite.. 
*)
FUNCTION_BLOCK DeviceWrite
VAR_INPUT
	En: 					BOOL;				(* Enable signal *)
	Instance: 				INT;				(* Instance is an address, use the function ToAddress() to convert station and device number to a valid address. *)
	Channel:				INT:=0;				(* Only used ff the device at the address has several channels. *)
	Data:	 				WORD;				(* The word to write to the device *)
	TimeOut:				TIME:=ComGVL.DEVICE_DEFAULT_TIME_OUT; (* Time out time to be used during read, default value is DEVICE_DEFAULT_TIME_OUT *)
END_VAR
VAR_OUTPUT
	Done:					BOOL:=FALSE;	(* If true, a data word was read ok, to reset set En to false *)
	Busy: 					BOOL:=FALSE;	(* Busy is true if the block is communicating with target, otherwise false. *)
	Error: 					BOOL:=FALSE;	(* True if any error, to reset error set En to low and then back to high*)
	ErrorID: 				COM_ERROR_VALUE:=COM_ERROR_VALUE.COM_ERR_NO_ERROR;	(* The error number, if no error the output is equal to COM_ERR_NO_ERROR i.e., 0 *)
	Sequence:				DEVICE_SEQUENCE;	(* Main Sequence for the function block. This output signal can be used for debug purposes. *)
	ErrorStep:				DEVICE_SEQUENCE;	(* Error step to help debug to where the error was. *)
END_VAR
VAR
	InstanceStatus:		INSTANCE_STATUS;
	AckWord:				WORD;
	fbTON_TimeOut: 		TON;
END_VAR

(* Check Instance status *)
InstanceStatus:=_GetInstance(Instance);
CASE InstanceStatus OF
	INSTANCE_STATUS.INSTANCE_STATUS_CANCEL:
		IF Sequence<> DEVICE_SEQUENCE.DEVICE_SEQUENCE_NOP AND Sequence<> DEVICE_SEQUENCE.DEVICE_SEQUENCE_TIME_OUT THEN
			Error:=TRUE;
			ErrorID:=COM_ERROR_VALUE.COM_ERR_CANCEL;
			Sequence:=DEVICE_SEQUENCE.DEVICE_SEQUENCE_CANCEL;
			_SetInstance(Instance, INSTANCE_STATUS.INSTANCE_STATUS_READY);
		END_IF;

 	INSTANCE_STATUS.INSTANCE_STATUS_FREE:									(* Device not allocated *)
		ErrorID:=COM_ERROR_VALUE.COM_ERR_NOT_ALLOCATED;
		Error:=TRUE;
		Busy:=FALSE;
		Done:=FALSE;
		Sequence:=DEVICE_SEQUENCE.DEVICE_SEQUENCE_NOP;
		RETURN;

	INSTANCE_STATUS.INSTANCE_STATUS_UNKNOWN:
		ErrorID:=COM_ERROR_VALUE.COM_ERR_LEVEL1;
		Error:=TRUE;
		Busy:=FALSE;
		Done:=FALSE;
		Sequence:=DEVICE_SEQUENCE.DEVICE_SEQUENCE_NOP;
		RETURN;
END_CASE;

(* Check if time out *)
IF fbTON_TimeOut.Q THEN
	NodeWriteStrobe(Instance, FALSE);
	NodeWriteWord(Instance, 0, 0);
	ErrorStep:=Sequence;
	Sequence:=DEVICE_SEQUENCE.DEVICE_SEQUENCE_TIME_OUT;
END_IF;

(* Main sequence *)
IF En THEN
	CASE Sequence OF
		DEVICE_SEQUENCE.DEVICE_SEQUENCE_TIME_OUT: (* -1, Error time out *)
			_SetInstance(Instance, INSTANCE_STATUS.INSTANCE_STATUS_READY);
			Busy:=FALSE;
			Done:=FALSE;
			Error:=TRUE;
			ErrorID:=COM_ERROR_VALUE.COM_ERR_LEVEL2_TIME_OUT;
			fbTON_TimeOut(IN:=FALSE);

		DEVICE_SEQUENCE.DEVICE_SEQUENCE_CANCEL: (* -2 *)
			Busy:=FALSE;
			Done:=FALSE;
			Error:=TRUE;
			ErrorID:=COM_ERROR_VALUE .COM_ERR_CANCEL;
			NodeWriteStrobe(Instance, FALSE);
			NodeWriteWord(Instance, 0, 0);

		DEVICE_SEQUENCE.DEVICE_SEQUENCE_ERROR: (* -3, Error during send/receive or GetStatus *)
			_SetInstance(Instance, INSTANCE_STATUS.INSTANCE_STATUS_READY);
			Busy:=FALSE;
			Done:=FALSE;
			Error:=TRUE;
			ErrorID:=COM_ERROR_VALUE.COM_ERR_LEVEL2_ERROR;
			fbTON_TimeOut(IN:=FALSE);

		DEVICE_SEQUENCE.DEVICE_SEQUENCE_NOP:
			ErrorId:=COM_ERROR_VALUE.COM_ERR_NO_ERROR;
			Error:=FALSE;
			IF NOT Done AND NOT Busy THEN
				IF InstanceStatus=INSTANCE_STATUS.INSTANCE_STATUS_READY THEN
					IF _SetInstance(Instance, INSTANCE_STATUS.INSTANCE_STATUS_BUSY) THEN
						Busy:=TRUE;
						Sequence:=DEVICE_SEQUENCE.DEVICE_SEQUENCE_INIT;
					END_IF;
				END_IF;
			END_IF;

		DEVICE_SEQUENCE.DEVICE_SEQUENCE_INIT: (* Init *)
			IF NOT NodeGetStatus(Instance) THEN
				ErrorStep:=Sequence;
				Sequence:=DEVICE_SEQUENCE.DEVICE_SEQUENCE_ERROR;
			ELSE
				Sequence:=DEVICE_SEQUENCE.DEVICE_SEQUENCE_WAIT_FOR_DEVICE_READY;
				NodeWriteStrobe(Instance, FALSE);
				NodeWriteWord(Instance, 0, 0);
			END_IF;

		DEVICE_SEQUENCE.DEVICE_SEQUENCE_WAIT_FOR_DEVICE_READY: (* Init of wait function *)
			fbTON_TimeOut(IN:=FALSE);
			Sequence:=DEVICE_SEQUENCE.DEVICE_SEQUENCE_WAIT_FOR_STROBE_LOW;

		DEVICE_SEQUENCE.DEVICE_SEQUENCE_WAIT_FOR_STROBE_LOW: (* Wait until target device is ready or time out *)
			fbTON_TimeOut(IN:=TRUE, PT:=TimeOut);
			IF NOT NodeReadStrobe(Instance) AND NodeReadWord(Instance, 0)=0 THEN
				fbTON_TimeOut(IN:=FALSE);
				Sequence:=DEVICE_SEQUENCE.DEVICE_SEQUENCE_PREPARE_SEND_RECEIVE;
			END_IF;

		DEVICE_SEQUENCE.DEVICE_SEQUENCE_PREPARE_SEND_RECEIVE:
			fbTON_TimeOut(IN:=FALSE);
			NodeWriteWord(Instance, 0, Data);
			Sequence:=DEVICE_SEQUENCE.DEVICE_SEQUENCE_STROBE_HIGH;

		DEVICE_SEQUENCE.DEVICE_SEQUENCE_STROBE_HIGH:
			NodeWriteStrobe(Instance, TRUE);
			Sequence:=DEVICE_SEQUENCE.DEVICE_SEQUENCE_SEND_RECEIVE;

		DEVICE_SEQUENCE.DEVICE_SEQUENCE_SEND_RECEIVE:  (*Wait for strobe high or time out *)
			fbTON_TimeOut(IN:=TRUE, PT:=TimeOut);

			IF NodeReadStrobe(Instance) THEN
				fbTON_TimeOut(IN:=FALSE);
				AckWord:=NodeReadWord(Instance, 0);
				NodeWriteWord(Instance, 0, 16#FFFF);

				IF AckWord=data THEN
	  				Sequence:=DEVICE_SEQUENCE.DEVICE_SEQUENCE_ACK;
				ELSE
					NodeWriteStrobe(Instance, FALSE);
					NodeWriteWord(Instance, 0, 0);
					ErrorStep:=Sequence;
	  				Sequence:=DEVICE_SEQUENCE.DEVICE_SEQUENCE_ERROR;
				END_IF;
			END_IF;

		DEVICE_SEQUENCE.DEVICE_SEQUENCE_ACK:
			NodeWriteStrobe(Instance, FALSE);
			Sequence:=DEVICE_SEQUENCE.DEVICE_SEQUENCE_WAIT_FOR_ANSWER;
			fbTON_TimeOut(IN:=FALSE);

		DEVICE_SEQUENCE.DEVICE_SEQUENCE_WAIT_FOR_ANSWER:
			fbTON_TimeOut(IN:=TRUE, PT:=TimeOut);
			IF NOT NodeReadStrobe(Instance) THEN
				fbTON_TimeOut(IN:=FALSE);
 				NodeWriteWord(Instance, 0, 0);
				Sequence:=DEVICE_SEQUENCE.DEVICE_SEQUENCE_SET_LOW;
			END_IF;

		DEVICE_SEQUENCE.DEVICE_SEQUENCE_SET_LOW:
			_SetInstance(Instance, INSTANCE_STATUS.INSTANCE_STATUS_READY);
			Busy:=FALSE;
			Sequence:=DEVICE_SEQUENCE.DEVICE_SEQUENCE_READY;

		DEVICE_SEQUENCE.DEVICE_SEQUENCE_READY:
			Done:=TRUE;
			(* Wait in this step until En=false *)

	END_CASE;
ELSE      (* En *)
	IF Busy THEN
		_SetInstance(Instance, INSTANCE_STATUS.INSTANCE_STATUS_READY);
	END_IF;

	Busy:=FALSE;
	Done:=FALSE;
	Error:=FALSE;
	ErrorId:=COM_ERROR_VALUE.COM_ERR_NOT_ENABLED;
	Sequence:=DEVICE_SEQUENCE.DEVICE_SEQUENCE_NOP;
END_IF; (* En *)

END_FUNCTION_BLOCK

// ---- ComLib/POUs/Private/_GetInstance.TcPOU
{library PRIVATE}
(*
  Private Funtcion:
  To get an Instance status.
*)
FUNCTION _GetInstance : INSTANCE_STATUS
VAR_INPUT
	Instance:			INT;				(* Instance, a number concatenated by SationNumber (1-INSTANCE_MAX_NUMBER_OF_STATIONS) and DeviceNumber (1-INSTANCE_MAX_NUMBER_OF_DEVICES). Instance is defined as: StaionNumber*100+DeviceNumber *)
END_VAR
VAR
	StationDevice: 	INT;
	StationNumber: 	INT;
END_VAR

_GetInstance:=INSTANCE_STATUS.INSTANCE_STATUS_UNKNOWN;

IF _CheckInstance(Instance) THEN
	StationNumber:=Instance/100;
	StationDevice:=Instance-StationNumber*100;
	_GetInstance:=ComGVL._Instance[StationNumber, StationDevice];
END_IF;

END_FUNCTION

// ---- ComLib/POUs/Private/_CheckInstance.TcPOU
{library PRIVATE}
(*
Private Funtcion:
Check if an Instance address is valid (within range) or not.
*)
FUNCTION _CheckInstance : BOOL
VAR_INPUT
	Instance: 			INT;			(* Instance, a number concatenated by SationNumber (1-INSTANCE_MAX_NUMBER_OF_STATIONS) and
                                                                       DeviceNumber (1-INSTANCE_MAX_NUMBER_OF_DEVICES). 
                                                                       Instance is defined as: StaionNumber*100+DeviceNumber *)
END_VAR
VAR
	StationNumber: 	INT;
	StationDevice: 	INT;
END_VAR

_CheckInstance:=FALSE;

IF Instance>=1*100 AND Instance<(ComGVL.INSTANCE_MAX_NUMBER_OF_STATIONS+1)*100 THEN
	StationNumber:=Instance/100;
	StationDevice:=Instance-StationNumber*100;

	IF StationDevice>0 AND StationDevice<= ComGVL.INSTANCE_MAX_NUMBER_OF_DEVICES THEN
		_CheckInstance:=TRUE;
	END_IF;
END_IF;

END_FUNCTION

// ---- ComLib/POUs/Private/_SetInstance.TcPOU
{library PRIVATE}
(*
  Private Funtcion:
  Set instance status.
*)

FUNCTION _SetInstance : BOOL
VAR_INPUT
	Instance: 				INT;		(* Instance, a number concatenated by SationNumber (1-INSTANCE_MAX_NUMBER_OF_STATIONS) and DeviceNumber (1-INSTANCE_MAX_NUMBER_OF_DEVICES). Instance is defined as: StaionNumber*100+DeviceNumber *)
	Status:					INSTANCE_STATUS;
END_VAR
VAR
	StationNumber: 		INT;
	StationDevice: 		INT;
END_VAR

_SetInstance:=FALSE;

IF _CheckInstance(Instance) THEN
	StationNumber:=Instance/100;
	StationDevice:=Instance-StationNumber*100;

	IF  ComGVL._Instance[StationNumber, StationDevice]<>INSTANCE_STATUS.INSTANCE_STATUS_FREE THEN
		ComGVL._Instance[StationNumber, StationDevice]:=Status;
		_SetInstance:=TRUE;
	END_IF;
END_IF;

END_FUNCTION

// ---- ComLib/POUs/Public/Level 1 Physical/NodeWriteStrobe.TcPOU
{library PUBLIC}
(* Level 1 function to write strobe value.
    Do not call this function from applications if functions on level 2-6 are used. *)
FUNCTION NodeWriteStrobe : BOOL
VAR_INPUT
	Address: 		INT;		(* Address, use the function ToAddress() to convert station and device number to a valid address. *)
	Value:			BOOL;		(* New strobe value. *)
END_VAR
VAR
	AWord:			WORD;
END_VAR

CASE NodeGetType(Address) OF
	DEVICE_TYPE.TYPE_ABB_1:  (* ABB Robot *)
		AWord:=ComGVL._qwABB;
		AWord.15:=Value;
		ComGVL._qwABB:=AWord;

	DEVICE_TYPE.TYPE_GANTRY_1:  (* Gantry robot *)
		AWord.15:=Value;
		(* Empty no real strobe *)


	DEVICE_TYPE.TYPE_SIMULATED:
		ComGVL._DataSimulatedStation[1, 1]:=BOOL_TO_BYTE(Value);
		AWord.15:=Value;
ELSE
		AWord:=0;
		AWord.15:=Value;
END_CASE;

(* Return value *)
NodeWriteStrobe:=AWord.15;

END_FUNCTION

// ---- ComLib/POUs/Public/Level 1 Physical/NodeGetType.TcPOU
{library PUBLIC}
(* Level 1 function to get communication type for a specific address.

   Depending on the address (specific device) different types of communication standards might exist.
   Note that this function does not transmit any data to check the real type of a device it only gives a predefined answer.
   On success the type is returned otherwise TYPE_ERROR.
*)

FUNCTION NodeGetType : DEVICE_TYPE
VAR_INPUT
	Address: INT;
END_VAR
VAR
END_VAR

CASE Address OF
	101, 201, 301, 401:  (* ABB robot *)
		NodeGetType:=DEVICE_TYPE.TYPE_ABB_1;

	502: (* Gantry robot *)
		NodeGetType:=DEVICE_TYPE.TYPE_GANTRY_1;

	ComGVL.ADDRESS_SIMULATED:  (* Simulated *)
		NodeGetType:=DEVICE_TYPE.TYPE_SIMULATED;

ELSE
		NodeGetType:=DEVICE_TYPE.TYPE_ERROR;
END_CASE;

END_FUNCTION

// ---- ComLib/POUs/Public/Level 1 Physical/NodeWriteWord.TcPOU
{library PUBLIC}
(* Level 1 function to write a word value.
    Do not call this function from applications if functions on level 2-6 are used. *)
FUNCTION NodeWriteWord : WORD
VAR_INPUT
	Address: 		INT;		(* Address, use the function ToAddress() to convert station and device number to a valid address. *)
	Channel:		INT:=0;		(* Only used ff the device at the address has several channels. *)
	Data:			WORD;		(* Data to write. *)
END_VAR
VAR
END_VAR

CASE NodeGetType(Address) OF
	DEVICE_TYPE.TYPE_ABB_1: (* ABB robot *)
		Data:=Data AND 16#7FFF;
		ComGVL._qwABB:=Data;

	DEVICE_TYPE.TYPE_GANTRY_1: (* Gantry robot *)
		Data:=Data AND 16#7FFF;

		CASE Channel OF
		0:
			ComGVL._qw1Gantry:=Data;
		1:
			ComGvl._qw2Gantry:=Data;
		2:
			ComGVL._qw3Gantry:=Data;
		ELSE
			Data:=0;
		END_CASE;

	DEVICE_TYPE.TYPE_SIMULATED:
		Data:=Data AND 16#7FFF;
		ComGVL._DataSimulatedStation[1, 2]:=WORD_TO_BYTE(Data);
ELSE
		Data:=0;
END_CASE;

(* Return value *)
NodeWriteWord:=Data;

END_FUNCTION

// ---- ComLib/POUs/Public/Level 1 Physical/NodeGetStatus.TcPOU
{library PUBLIC}
(* Level 1 function to get communication status for a specific address.

   Depending on the address (specific device) different status checks can be performed, e.g., bus status.
   Note that this function does not transmit any data to check the real status of a device it only check if it is possible to communicate.
   On success true is returned otherwise false.
*)
FUNCTION NodeGetStatus : BOOL
VAR_INPUT
	Address: 		INT;		(* Address, use the function ToAddress() to convert station and device number to a valid address. *)
END_VAR
VAR
END_VAR

NodeGetStatus:=FALSE;

IF _CheckInstance(Address) THEN
	NodeGetStatus:=TRUE;

	(* Code here to check bus status *)
END_IF;

END_FUNCTION

// ---- ComLib/POUs/Public/Level 1 Physical/NodeReadStrobe.TcPOU
{library PUBLIC}
(* Level 1 function to read strobe value.
    Do not call this function from applications if functions on level 2-6 are used. *)
FUNCTION NodeReadStrobe : BOOL
VAR_INPUT
	Address: 		INT;		(* Address, use the function ToAddress() to convert station and device number to a valid address. *)
END_VAR
VAR
	wAbb: 					WORD;
	StrobeValue:			BOOL;
	_DataStation500: BOOL;
END_VAR

CASE NodeGetType(Address) OF
	DEVICE_TYPE.TYPE_ABB_1:  	(* ABB robot *)
		wAbb:=ComGVL._iwABB;		(* Note: Direct access to input data *)
		StrobeValue:=wAbb.15;

	DEVICE_TYPE.TYPE_GANTRY_1: 	(* Gantry robot *)
		StrobeValue:=0;

	DEVICE_TYPE.TYPE_SIMULATED:
		StrobeValue:=BYTE_TO_BOOL(ComGVL._DataSimulatedStation[2, 1]);

ELSE
		StrobeValue:=FALSE;
END_CASE;

(* Return value *)
NodeReadStrobe:=StrobeValue;

END_FUNCTION

// ---- ComLib/POUs/Public/Level 1 Physical/NodeReadWord.TcPOU
{library PUBLIC}
(* Llevel 1 function to read a word value.
    Do not call this function from applications if functions on level 2-6 are used. *)
FUNCTION NodeReadWord : WORD
VAR_INPUT
	Address: 		INT;		(* Address, use the function ToAddress() to convert station and device number to a valid address. *)
	Channel:		INT:=0;		(* Only used ff the device at the address has several channels. *)
END_VAR
VAR
	Data:			WORD;
	wAbb:			WORD;
	wGantry:		WORD;
END_VAR

CASE NodeGetType(Address) OF
	DEVICE_TYPE.TYPE_ABB_1: 	(* ABB robot *)
		wAbb:=ComGVL._iwABB;		(* Note: Direct access to input data *)
		Data:=wAbb AND 16#7FFF; (* Filter to remove strobe signal *)

	DEVICE_TYPE.TYPE_GANTRY_1: 	(* Gantry robot *)
		CASE Channel OF
		0:
			wGantry:=ComGVL._iw1Gantry;
		1:
			wGantry:=ComGVL._iw2Gantry;
		2:
			wGantry:=ComGVL._iw3Gantry;
		ELSE
			Data:=0;
		END_CASE;

		Data:=wGantry AND 16#7FFF;	 (* Filter to remove strobe signal *)

	DEVICE_TYPE.TYPE_SIMULATED:
		Data:=BYTE_TO_WORD(ComGVL._DataSimulatedStation[2, 2]);

ELSE
		Data:=0;
END_CASE;

(* Return value *)
NodeReadWord:=Data;

END_FUNCTION

// ---- ComLib/POUs/Public/Level 2 Data link/DeviceRead.TcPOU
{library PUBLIC}
(*
  Function to read a word from a specific device defined by Instance number.
  The Instance must be open (DeviceOpen or DeviceUse) before you can use DeviceRead. 
*)
FUNCTION_BLOCK DeviceRead
VAR_INPUT
	En: 					BOOL;				(* Enable signal *)
	Instance: 				INT;				(* Instance is an address, use the function ToAddress() to convert station and device number to a valid address. *)
	Channel:				INT:=0;				(* Only used ff the device at the address has several channels. *)
	TimeOut:				TIME:=ComGVL.DEVICE_DEFAULT_TIME_OUT; (* Time out time to be used during read, default value is DEVICE_DEFAULT_TIME_OUT *)
END_VAR
VAR_OUTPUT
	Done:					BOOL:=FALSE;		(* If true, a data word was read ok, to reset set En to false *)
	Busy: 					BOOL:=FALSE;		(* Busy is true if the block is communicating with target, otherwise false. *)
	Error: 					BOOL:=FALSE;		(* True if any error, to reset error set En to low and then back to high*)
	ErrorID: 				COM_ERROR_VALUE:=COM_ERROR_VALUE.COM_ERR_NO_ERROR;	(* The error number, if no error the output is equal to COM_ERR_NO_ERROR i.e., 0 *)
	Data:	 				WORD;				(* The word read from the device *)
	Sequence:				DEVICE_SEQUENCE;	(* Main Sequence for the function block. This output signal can be used for debug purposes. *)
	ErrorStep:				DEVICE_SEQUENCE;	(* Error step to help debug to where the error was. *)
END_VAR
VAR
	InstanceStatus:		INSTANCE_STATUS;
	fbTON_TimeOut: 		TON;
END_VAR

(* Check Instance status *)
InstanceStatus:=_GetInstance(Instance);
CASE InstanceStatus OF
	INSTANCE_STATUS.INSTANCE_STATUS_CANCEL:
		IF Sequence<> DEVICE_SEQUENCE.DEVICE_SEQUENCE_NOP AND Sequence<> DEVICE_SEQUENCE.DEVICE_SEQUENCE_TIME_OUT THEN
			Error:=TRUE;
			ErrorID:=COM_ERROR_VALUE.COM_ERR_CANCEL;
			Sequence:=DEVICE_SEQUENCE.DEVICE_SEQUENCE_CANCEL;
			_SetInstance(Instance, INSTANCE_STATUS.INSTANCE_STATUS_READY);
		END_IF;

 	INSTANCE_STATUS.INSTANCE_STATUS_FREE:									(* Device not allocated *)
		ErrorID:=COM_ERROR_VALUE.COM_ERR_NOT_ALLOCATED;
		Error:=TRUE;
		Busy:=FALSE;
		Done:=FALSE;
		Sequence:=DEVICE_SEQUENCE.DEVICE_SEQUENCE_NOP;
		RETURN;

	INSTANCE_STATUS.INSTANCE_STATUS_UNKNOWN:
		ErrorID:=COM_ERROR_VALUE.COM_ERR_LEVEL1;
		Error:=TRUE;
		Busy:=FALSE;
		Done:=FALSE;
		Sequence:=DEVICE_SEQUENCE.DEVICE_SEQUENCE_NOP;
		RETURN;
END_CASE;

(* Check if time out *)
IF fbTON_TimeOut.Q THEN
	NodeWriteStrobe(Instance, FALSE);
	NodeWriteWord(Instance, 0, 0);
	ErrorStep:=Sequence;
	Sequence:=DEVICE_SEQUENCE.DEVICE_SEQUENCE_TIME_OUT;
END_IF;

(* Main sequence *)
IF En THEN
	CASE Sequence OF
		DEVICE_SEQUENCE.DEVICE_SEQUENCE_TIME_OUT: (* -1, Error time out *)
			_SetInstance(Instance, INSTANCE_STATUS.INSTANCE_STATUS_READY);
			Busy:=FALSE;
			Done:=FALSE;
			Error:=TRUE;
			ErrorID:=COM_ERROR_VALUE .COM_ERR_NO_ERROR;
			fbTON_TimeOut(IN:=FALSE);

		DEVICE_SEQUENCE.DEVICE_SEQUENCE_CANCEL:
			Busy:=FALSE;
			Done:=FALSE;
			Error:=TRUE;
			ErrorID:=COM_ERROR_VALUE.COM_ERR_CANCEL;
			NodeWriteStrobe(Instance, FALSE);
			NodeWriteWord(Instance, 0, 0);

		DEVICE_SEQUENCE.DEVICE_SEQUENCE_ERROR: (* -3, Error during send/receive or GetStatus  *)
			_SetInstance(Instance, INSTANCE_STATUS.INSTANCE_STATUS_READY);
			Busy:=FALSE;
			Done:=FALSE;
			Error:=TRUE;
			ErrorID:=COM_ERROR_VALUE.COM_ERR_LEVEL2_ERROR;
			fbTON_TimeOut(IN:=FALSE);

		DEVICE_SEQUENCE.DEVICE_SEQUENCE_NOP:
			ErrorId:=COM_ERROR_VALUE.COM_ERR_NO_ERROR;
			Error:=FALSE;
			IF NOT Done AND NOT Busy THEN
				IF InstanceStatus=INSTANCE_STATUS.INSTANCE_STATUS_READY THEN
					IF _SetInstance(Instance, INSTANCE_STATUS.INSTANCE_STATUS_BUSY) THEN
						Busy:=TRUE;
						Sequence:=DEVICE_SEQUENCE.DEVICE_SEQUENCE_INIT;
					END_IF;
				END_IF;
			END_IF;

		DEVICE_SEQUENCE.DEVICE_SEQUENCE_INIT: (* Init *)
			IF NOT NodeGetStatus(Instance) THEN
				ErrorStep:=Sequence;
				Sequence:=Sequence:=DEVICE_SEQUENCE.DEVICE_SEQUENCE_ERROR;
			ELSE
				Sequence:=DEVICE_SEQUENCE.DEVICE_SEQUENCE_WAIT_FOR_DEVICE_READY;
				NodeWriteStrobe(Instance, FALSE);
				NodeWriteWord(Instance, 0, 0);
			END_IF;

		DEVICE_SEQUENCE.DEVICE_SEQUENCE_WAIT_FOR_DEVICE_READY: (* Init of wait function *)
			fbTON_TimeOut(IN:=FALSE);
			Sequence:=DEVICE_SEQUENCE.DEVICE_SEQUENCE_WAIT_FOR_STROBE_LOW;

		DEVICE_SEQUENCE.DEVICE_SEQUENCE_WAIT_FOR_STROBE_LOW:
			Sequence:=DEVICE_SEQUENCE.DEVICE_SEQUENCE_PREPARE_SEND_RECEIVE;

		DEVICE_SEQUENCE.DEVICE_SEQUENCE_PREPARE_SEND_RECEIVE:
			fbTON_TimeOut(IN:=FALSE);
			Sequence:=DEVICE_SEQUENCE.DEVICE_SEQUENCE_STROBE_HIGH;

		DEVICE_SEQUENCE.DEVICE_SEQUENCE_STROBE_HIGH: (*Wait for strobe high or time out *)
			fbTON_TimeOut(IN:=TRUE, PT:=TimeOut);

			IF NodeReadStrobe(Instance) THEN
				Sequence:=DEVICE_SEQUENCE.DEVICE_SEQUENCE_SEND_RECEIVE;
				fbTON_TimeOut(IN:=FALSE);
			END_IF;

		DEVICE_SEQUENCE.DEVICE_SEQUENCE_SEND_RECEIVE:
			Data:=NodeReadWord(Instance, 0);
			NodeWriteWord(Instance, 0, Data);
  			Sequence:=DEVICE_SEQUENCE.DEVICE_SEQUENCE_ACK;

		DEVICE_SEQUENCE.DEVICE_SEQUENCE_ACK:
			NodeWriteStrobe(Instance, TRUE);
			Sequence:=DEVICE_SEQUENCE.DEVICE_SEQUENCE_WAIT_FOR_ANSWER;
			fbTON_TimeOut(IN:=FALSE);

		DEVICE_SEQUENCE.DEVICE_SEQUENCE_WAIT_FOR_ANSWER:
			fbTON_TimeOut(IN:=TRUE, PT:=TimeOut);
			IF NOT NodeReadStrobe(Instance) THEN
				NodeWriteStrobe(Instance, FALSE);

				fbTON_TimeOut(IN:=FALSE);
				Sequence:=DEVICE_SEQUENCE.DEVICE_SEQUENCE_SET_LOW;
			END_IF;

		DEVICE_SEQUENCE.DEVICE_SEQUENCE_SET_LOW:
			NodeWriteWord(Instance, 0, 0);

			_SetInstance(Instance, INSTANCE_STATUS.INSTANCE_STATUS_READY);
			Busy:=FALSE;
			Sequence:=DEVICE_SEQUENCE.DEVICE_SEQUENCE_READY;

		DEVICE_SEQUENCE.DEVICE_SEQUENCE_READY:
			Done:=TRUE;
			(* Wait in this step until En=false *)

	END_CASE;
ELSE      (* En *)
	IF Busy THEN
		_SetInstance(Instance, INSTANCE_STATUS.INSTANCE_STATUS_READY);
	END_IF;

	Busy:=FALSE;
	Done:=FALSE;
	Error:=FALSE;
	ErrorId:=COM_ERROR_VALUE.COM_ERR_NOT_ENABLED;
	Sequence:=DEVICE_SEQUENCE.DEVICE_SEQUENCE_NOP;
END_IF; (* En *)

END_FUNCTION_BLOCK

// ---- ComLib/POUs/Public/Level 2 Data link/DeviceCancel.TcPOU
{library PUBLIC}
(* Use this function to cancel an ongoing communication action to a specific device defined by Instance *)
FUNCTION_BLOCK DeviceCancel
VAR_INPUT
	En:						BOOL;		(* Enable signal *)
	Instance: 				INT;		(* Instance is an aAddress, use the function ToAddress() to convert station and device number to a valid address. *)
END_VAR
VAR_OUTPUT
	Done: 					BOOL;		(* True if En is true *)
END_VAR

IF En THEN
	IF _GetInstance(Instance)=INSTANCE_STATUS.INSTANCE_STATUS_BUSY THEN
		_SetInstance(Instance, INSTANCE_STATUS.INSTANCE_STATUS_CANCEL);
	END_IF;

	Done:=TRUE;

ELSE
	Done:=FALSE;
END_IF;

END_FUNCTION_BLOCK

// ---- ComLib/POUs/Public/Level 2 Data link/DeviceOpen.TcPOU
{library PUBLIC}
(* Use this function to open an communication link to a specific device defined by Instance.
A communication link is always opened for read/write.
Return value is true if open was ok otherwise false. *)
FUNCTION DeviceOpen : BOOL
VAR_INPUT
	Instance: 				INT;		(* Instance is an address, use the function ToAddress() to convert station and device number to a valid address. *)
END_VAR

DeviceOpen:=FALSE;
IF _GetInstance(Instance)=INSTANCE_STATUS.INSTANCE_STATUS_FREE THEN
	IF _CheckInstance(Instance) THEN
		IF _AllocateInstance(Instance) THEN
			DeviceOpen:=TRUE;
		END_IF;
	END_IF;
END_IF;

END_FUNCTION

// ---- ComLib/POUs/Private/_AllocateInstance.TcPOU
{library PRIVATE}
(*
  Private Funtcion:
  Allocates a communications instance.

  Return true if station is available for allocation. 
*)

FUNCTION _AllocateInstance : BOOL
VAR_INPUT
	Instance: 				INT;		(* Instance, a number concatenated by SationNumber (1-INSTANCE_MAX_NUMBER_OF_STATIONS) and DeviceNumber (1-INSTANCE_MAX_NUMBER_OF_DEVICES). Instance is defined as: StaionNumber*100+DeviceNumber *)
END_VAR
VAR
	StationNumber: 		INT;
	StationDevice: 		INT;
END_VAR

_AllocateInstance:=FALSE;

IF _CheckInstance(Instance) THEN
	StationNumber:=Instance/100;
	StationDevice:=Instance-StationNumber*100;

	IF  ComGVL._Instance[StationNumber, StationDevice]= INSTANCE_STATUS.INSTANCE_STATUS_FREE THEN
		ComGVL._Instance[StationNumber, StationDevice]:=INSTANCE_STATUS.INSTANCE_STATUS_READY;
		_AllocateInstance:=TRUE;
	END_IF;
END_IF;

END_FUNCTION

// ---- ComLib/POUs/Public/Level 4 Transport/DatagramCheckSum.TcPOU
{library PUBLIC}
(* This function will return the checksum for a specific DataGram message.
  Note: the DataGram is not changed including the CheckSum member by this function, only calculated.
  You need to set the correct value in the DataGram.*)
FUNCTION DatagramCheckSum : BYTE
VAR_INPUT
	Data:		DataGram;
END_VAR
VAR
	Ptr: 		POINTER TO BYTE;
	Size: 		INT;
	i: 			INT;
	CkSum: 	BYTE;
END_VAR

Size:=_DataGramSize()-1;

CkSum:=0;
Ptr:=ADR(Data);

FOR i:=1 TO Size DO
	CkSum:=CkSum+Ptr^;
	Ptr:=Ptr+1;
END_FOR;

DatagramCheckSum:=CkSum;

END_FUNCTION

// ---- ComLib/POUs/Private/_DataGramSize.TcPOU
{library PRIVATE}
(*
  Private Funtcion:
  Get the size for a datagram struct. The SIZEOF operator does not work on all systems. In all cases this function is safer.
*)
FUNCTION _DataGramSize : INT  
VAR_INPUT
END_VAR
VAR
	Data: 	DataGram;
END_VAR

 _DataGramSize:=SIZEOF(Data);
  
(* Enable this row if SIZEOF() does not work *)
(* _DataGramSize:=8; *)

END_FUNCTION

// ---- ComLib/POUs/Public/Level 6 Presentation/ABB/Goto/ABBGoToHome.TcPOU
{library PUBLIC}
(* Function to send a robot to home location *)
FUNCTION_BLOCK ABBGoToHome
VAR_INPUT
	En: 			BOOL:=FALSE;				(* Set to true to start *)
END_VAR
VAR_OUTPUT
	Done: 				BOOL:=FALSE;			(* If true, the command is transmitted ok, to reset set En to false *)
	Executing:			BOOL:=FALSE;			(* True while the command in transmitted *)
	Waiting:			BOOL:=FALSE;			(* True if the command is queued to be transmitted *)
	Error: 				BOOL := FALSE;			(* True if an error occured *)
	Progress:			INT:=0;						(* Function progress *)
END_VAR
VAR_IN_OUT
	Data: 				CommunicationData;		(* Common data structure to connect this function block to a specific Communicator block *)
END_VAR
VAR
	FunctionType: 		FUNCTION_TYPE;
	FunctionNumber: 	INT;
	ParameterDW:	DWORD;
	ParameterB:		BYTE;
	Sequence:			INT:=0;

	fbRPC:				ASyncRPC;
END_VAR

FunctionType:=FUNCTION_TYPE.FUNCTION_TYPE_ASYNC_RPC;
FunctionNumber:=ABB_ASYNC_FUNCTION_GOTO_HOME;
ParameterDW:=0;										(* No parameters *)
ParameterB:=0;

fbRPC(EN:=En, Data:=Data, FunctionType:=FunctionType,FunctionNumber:=FunctionNumber, ParameterDW:=ParameterDW, ParameterB:=ParameterB);

Done:=fbRPC.Done;
Executing:=fbRPC.Executing;
Waiting:=fbRPC.Waiting;
Error:=fbRPC.Error OR (fbRPC.Done AND fbRPC.ReturnValue<0);
Progress:=fbRPC.Progress;

END_FUNCTION_BLOCK

// ---- ComLib/POUs/Public/Level 5 Session/RPC Remote Procedural Call/ASyncRPC.TcPOU
{library PUBLIC}
(*
ASyncRPC will handle ASync RPC calls with 1 parameter.
It is possible to use RPC1 to start a ASync call however, ASyncRPC will wait until the function call is done.

A session will be established to the specific equipment during the function call and when a return value (or error) the session is ended.
It is possible to queue many calls by cascade coupled blocks in serie or parallel.

By using the Done output signal as input to En on another function block it is possible to serialise calls.

*)
FUNCTION_BLOCK ASyncRPC
VAR_INPUT
	En: 				BOOL:=FALSE;				(* Set to true to call a  RPC function and wait for an answer *)
	FunctionType:		FUNCTION_TYPE:=FUNCTION_TYPE.FUNCTION_TYPE_ASYNC_RPC;			(* Function type set to  ASYNC *)
	FunctionNumber:	INT;							(* RPC function number *)
	ParameterDW:	DWORD;							(* DWORD parameter value *)
	ParameterB:		BYTE;							(* Byte parameter value *)
END_VAR
VAR_OUTPUT
	Done: 				BOOL:=FALSE;				(* If true, the command is transmitted ok, to reset set En to false *)
	Executing:			BOOL:=FALSE;				(* True while the command in transmitted *)
	Waiting:			BOOL:=FALSE;				(* True if the command is queued to be transmitted *)
	Error: 				BOOL := FALSE;				(* True if an communication error occured *)
	Progress:			INT:=0;							(* Async progress *)
	ReturnValue:		FUNCTION_TYPE;				(* Return value, negative i.e. FUNCTION_TYPE_ERROR_NO_FUNCTION is an error error *)
END_VAR
VAR_IN_OUT
	Data: 				CommunicationData;			(* Common data structure to connect this function block to a specific Communicator block *)
END_VAR
VAR
	fbSessionInit: 	 SessionInit;
	fbSessionSend: 	 SessionSend;
	fbSessionStatus: SessionSend;
	fbSessionEnd: 	 SessionEnd;
	Sequence:			INT:=0;
	ReStart:			BOOL:=FALSE;
	Ended:				BOOL:=FALSE;
	RetMem: 			BYTE;
END_VAR

//IF fbSessionInit.Done AND NOT fbSessionInit.Established AND En THEN
// fbSessionInit(En:=FALSE, Data:=Data);
//ELSE
 fbSessionInit(En:=En, Data:=Data); 
//END_IF

fbSessionSend(En:=fbSessionInit.Done, SessionID:=fbSessionInit.SessionID, Data:=Data,
                             FunctionType:=INT_TO_BYTE(FunctionType), FunctionNumber:=INT_TO_BYTE(FunctionNumber), 
									ParameterDW:=ParameterDW, ParameterB:=ParameterB);

fbSessionStatus(En:=fbSessionInit.Done AND NOT ReStart, SessionID:=fbSessionInit.SessionID, Data:=Data,
                             FunctionType:=INT_TO_BYTE(FUNCTION_TYPE.FUNCTION_TYPE_INFORMATION), 
								FunctionNumber:=INT_TO_BYTE(INFO_FUNCTION_NUMBER.INFO_FUNCTION_RPC_STATUS), 
										ParameterDW:=0, ParameterB:=0);

fbSessionEnd(En:=fbSessionStatus.Done AND Ended, SessionID:=fbSessionInit.SessionID, Data:=Data);

IF NOT En THEN
	Sequence:=0;
	Progress:=0;
	Ended:=FALSE;
END_IF;

CASE Sequence OF
0:		(* Wait for function to start *)
		Done:=FALSE;
		Progress:=0;
		Executing:=fbSessionSend.Executing;
		Waiting:=fbSessionSend.Waiting;
		Error:=fbSessionSend.Error;
		Ended:=FALSE;
		ReturnValue:=FUNCTION_TYPE.FUNCTION_TYPE_ASYNC_RPC; (* Default value *)

		IF fbSessionSend.Error THEN
			ReturnValue:=FUNCTION_TYPE.FUNCTION_TYPE_ERROR_NO_FUNCTION;
			Sequence:=100;
		ELSIF fbSessionSend.Done THEN
			Sequence:=10;
		END_IF;

10:		(* Check if any error during start of function *)
		IF fbSessionSend.Answer.FunctionType<0 THEN
			ReturnValue:=FUNCTION_TYPE.FUNCTION_TYPE_ERROR_NO_FUNCTION;
			Sequence:=100;
		ELSE
			Data._ASyncProgress:=Progress;
			Sequence:=20;
		END_IF;

20:		(* Ask for status *)
		Done:=FALSE;
		Executing:=fbSessionStatus.Executing;
		Waiting:=fbSessionStatus.Waiting;
		Error:=fbSessionStatus.Error;

		IF fbSessionStatus.Error THEN
			ReturnValue:=FUNCTION_TYPE.FUNCTION_TYPE_ERROR_NO_FUNCTION;
			Sequence:=100;
		ELSIF fbSessionStatus.Done THEN
			Sequence:=30;
		END_IF;

30:		(* Check for any error during call for status *)
		IF fbSessionStatus.Answer.FunctionType<0 THEN  (* This is true if the status call does not exist in the device *)
			ReturnValue:=fbSessionStatus.Answer.FunctionType;   				
			Sequence:=100;
		ELSE
			Progress:=DWORD_TO_INT((SHR(fbSessionStatus.Answer.ParameterDW, 24) AND  16#FF));
			Data._ASyncProgress:=Progress;
			Data._ASyncStatus:=_GetStatusInformation(fbSessionStatus.Answer);
			Data._ASyncStatusCounter:=Data._ASyncStatusCounter+1;
			Sequence:=40;
		END_IF;

40:		(* Check if status call is ready or error *)
		RetMem:=DWORD_TO_BYTE((SHR(fbSessionStatus.Answer.ParameterDW, 8) AND  16#FF));
		IF ((DWORD_TO_BYTE(fbSessionStatus.Answer.ParameterDW) AND 16#FF)=0) THEN
			IF RetMem=16#FF THEN (* This is true if the RPC function does not exist *)
				ReturnValue:=FUNCTION_TYPE.FUNCTION_TYPE_ERROR_NO_FUNCTION;
				Sequence:=100;
			ELSE
				Sequence:=80;
			END_IF;
		ELSE
			Sequence:=50;
		END_IF;

50:		(* Restart status question *)
		ReStart:=TRUE;
		Sequence:=60;

60:		(* Restart done *)
		ReStart:=FALSE;
		Sequence:=20;

80:		(* ASyncRPC Done *)
		Progress:=100;
		Data._ASyncProgress:=Progress;

		Done:=fbSessionStatus.Done;
		Executing:=fbSessionStatus.Executing;
		Waiting:=fbSessionStatus.Waiting;
		Error:=fbSessionStatus.Error;
		ReturnValue:=FunctionType;
		Ended:=TRUE;

100:	(* Error *)
		Done:=FALSE;
		Executing:=FALSE;
		Waiting:=FALSE;
		Error:=TRUE;
END_CASE;

END_FUNCTION_BLOCK

// ---- ComLib/POUs/Public/Level 5 Session/Session/SessionInit.TcPOU
{library PUBLIC}
(* Use this function block to initiate, maintain and end a session. The session is queued
    when En=TRUE, when a session is possible Established is set to True. If En becomes FALSE and the a session is queued (waiting) the 
    session is aborted. However, if a session is established ongoing transmistion is not aborted.  To abort an ongoing transmission set En to FALSE 
   and disable the he Communicator block (En=FALSE) at the same time.
*)
FUNCTION_BLOCK SessionInit
VAR_INPUT
	En:					BOOL:=FALSE;			(* Set to true to Initiate and maintain a session and to end a session or abort set to low *)
END_VAR
VAR_OUTPUT
	Done:				BOOL:=FALSE;			(* Set to true when En is true and a session is established, set to false when En is false *)
	Established:		BOOL:=FALSE;			(* True if a session is established *)
	SessionID:		INT:=-1;					(* A  session ID number or -1 if no active session *)
END_VAR
VAR_IN_OUT
	Data: 				CommunicationData;		(* Common data structure to connect this function block to a specific Communicator block *)
END_VAR
VAR
	Sequence: 		INT := 0;
END_VAR

IF En THEN
	CASE Sequence OF
		0: (* Wait until possible to get a session *)
			IF NOT Data._Session._Locked AND Data._Status=DATAGRAM_SEQUENCE.DATAGRAM_SEQUENCE_NOP AND Data._DataExecute=Data._DataCounter THEN
				Data._Session._Locked:=TRUE;
				Data._Session._SessionID:=Data._Session._SessionID+1;
				Data._Session._SessionCounter:=0;
				Data._Session._SessionBussy:=FALSE;
				Data._DataExecute:=0;
				Data._DataCounter:=0;

				SessionID:=Data._Session._SessionID;
				Established:=TRUE;
				Done:=TRUE;
				Sequence:=1;
			END_IF;

		1:
			(* Some one else has closed the session *)
			IF NOT Data._Session._Locked OR SessionID<>Data._Session._SessionID THEN
				Established:=FALSE;
				SessionID:=-1;
			END_IF;
	END_CASE;
ELSE
	Sequence:=0;
	Done:=FALSE;
 	IF Established THEN
		Data._Session._Locked:=FALSE;
		Established:=FALSE;
		SessionID:=-1;
	END_IF;
END_IF;

END_FUNCTION_BLOCK

// ---- ComLib/POUs/Public/Level 5 Session/Session/SessionSend.TcPOU
{library PUBLIC}
(*
Use this function block to send DataGram to a equipment.
To send a Session must exist, use SessionInit to create a session.
*)
FUNCTION_BLOCK SessionSend
VAR_INPUT
	En:				BOOL;						(* Set to true to send a data gram *)
	SessionID: 		INT;					 	(* A  valid session ID number generated by SessionInit *)
	FunctionType:	BYTE;						(* Function type ASYNC or SYNC *)
	FunctionNumber:	BYTE;						(* Function number *)
	ParameterDW:	DWORD;						(* DWORD parameter value *)
	ParameterB:		BYTE;						(* Byte parameter value *)
END_VAR
VAR_OUTPUT
	Done: 				BOOL:=FALSE;			(* If true, the command is transmitted ok, to reset set En to false *)
	Executing:			BOOL:=FALSE;			(* True while the command in transmitted *)
	Waiting:			BOOL:=FALSE;			(* True if the command is queued to be transmitted *)
	Error: 				BOOL := FALSE;			(* True if an error occured *)
	Answer:	 			DataGram;				(* Answer from send *)
	BytesLeft:			INT;					(* Number of bytes left to send *)
END_VAR
VAR_IN_OUT
	Data: 				CommunicationData;		(* Common data structure to connect this function block to a specific Communicator block *)
END_VAR
VAR
	Sequence:		INT:=0;
	MySession:	INT:=-1;
END_VAR

IF  En THEN
	IF  SessionID=Data._Session._SessionID AND SessionID<>-1 AND Data._Session._Locked THEN
		CASE Sequence OF
			0:	(* Wait until ready *)
				Waiting:=TRUE;
				BytesLeft:=_DataGramSize();
				IF Data._Status=DATAGRAM_SEQUENCE.DATAGRAM_SEQUENCE_NOP AND NOT Data._Session._SessionBussy THEN
					Waiting:=FALSE;
					Data._Session._SessionBussy:=TRUE;
					Sequence:=Sequence+1;
				END_IF;

			1:	(* Copy data to send buffer *)
				Data._Data.FunctionType:=FunctionType;
				Data._Data.FunctionNumber:=FunctionNumber;
				Data._Data.ParameterDW:=ParameterDW;
				Data._Data.ParameterB:=ParameterB;

				MySession:=Data._Session._SessionCounter;
				Data._DataExecute:= Data._DataCounter+INT_TO_UDINT(_DataGramSize());
				BytesLeft:=_DataGramSize();
				Executing:=TRUE;
				Sequence:=Sequence+1;

			2:	(* Wait until all data send *)
 				BytesLeft:=UDINT_TO_INT(Data._DataExecute-Data._DataCounter);

				IF Data._Error THEN
					Data._Session._SessionBussy:=FALSE;
					Error:=TRUE;
					Sequence:=Sequence+1;
				ELSIF Data._Session._SessionCounter<>MySession THEN
					Data._Session._SessionBussy:=FALSE;
					Answer:=Data._DataAnswer;
					Done:=TRUE;
					Sequence:=Sequence+1;
				END_IF;

			3:
				Waiting:=FALSE;
				Executing:=FALSE;
		END_CASE;
	ELSE
		Waiting:=FALSE;
		Executing:=FALSE;
		Sequence:=0;
	END_IF;
ELSE
	Done:=FALSE;
	Waiting:=FALSE;
	Executing:=FALSE;
	Error:=FALSE;
	BytesLeft:=0;
	Sequence:=0;
END_IF;

END_FUNCTION_BLOCK

// ---- ComLib/POUs/Public/Level 5 Session/Session/SessionEnd.TcPOU
{library PUBLIC}
(* Use this function block to end an ongoing session. This is the same thing as setting En to false on the SessionInit block,
   An ongoing transmistion is not aborted.  To abort an ongoing transmission set En to TRUE
   and disable the he Communicator block (En=FALSE) at the same time.
*)
FUNCTION_BLOCK SessionEnd
VAR_INPUT
	En:					BOOL:=FALSE;			(* Set to true to end a session *)
	SessionID:		INT:=-1;					(* A  valid session ID number generated by SessionInit *)
END_VAR
VAR_OUTPUT
	Done:				 BOOL;						(* True if session was ended *)
END_VAR
VAR_IN_OUT
	Data: 				CommunicationData;		(* Common data structure to connect this function block to a specific Communicator block *)
END_VAR

IF En THEN
	IF SessionId<>-1 THEN
		IF SessionID=Data._Session._SessionID AND  Data._Session._Locked THEN
			Data._Session._Locked:=FALSE;
			Done:=TRUE;
		END_IF;
	END_IF;
ELSE
	Done:=FALSE;
END_IF;

END_FUNCTION_BLOCK

// ---- ComLib/POUs/Private/_GetStatusInformation.TcPOU
{library PRIVATE}
(*
  Private Funtcion:
  Decode Status information messages.

*)
FUNCTION _GetStatusInformation : StatusInformationData
VAR_INPUT
	Data: 				DataGram;
END_VAR
VAR
END_VAR

_GetStatusInformation.Progress:=DWORD_TO_INT((SHR(Data.ParameterDW, 24) AND  16#FF));
_GetStatusInformation.FunctionNumber:=BYTE_TO_INT(Data.FunctionNumber);
_GetStatusInformation.ReturnValue:=BYTE_TO_INT(Data.FunctionType);
_GetStatusInformation.Extra:=BYTE_TO_INT(Data.ParameterB);

END_FUNCTION

// ---- ComLib/POUs/Public/Level 6 Presentation/ABB/Goto/ABBGoToTable.TcPOU
{library PUBLIC}
(* Function to send a robot to storage location *)
FUNCTION_BLOCK ABBGoToTable
VAR_INPUT
	En: 			BOOL:=FALSE;				(* Set to true to start *)
END_VAR
VAR_OUTPUT
	Done: 				BOOL:=FALSE;			(* If true, the command is transmitted ok, to reset set En to false *)
	Executing:			BOOL:=FALSE;			(* True while the command in transmitted *)
	Waiting:			BOOL:=FALSE;			(* True if the command is queued to be transmitted *)
	Error: 				BOOL := FALSE;			(* True if an error occured *)
	Progress:			INT:=0;						(* Function progress *)
END_VAR
VAR_IN_OUT
	Data: 				CommunicationData;		(* Common data structure to connect this function block to a specific Communicator block *)
END_VAR
VAR
	FunctionType: 		FUNCTION_TYPE;
	FunctionNumber: 	INT;
	ParameterDW:		DWORD;
	ParameterB:			BYTE;
	Sequence:			INT:=0;

	fbRPC:				ASyncRPC;
END_VAR

FunctionType:=FUNCTION_TYPE.FUNCTION_TYPE_ASYNC_RPC;
FunctionNumber:=ABB_ASYNC_FUNCTION_GOTO_TABLE;
ParameterDW:=0;										(* No parameters *)
ParameterB:=0;

fbRPC(EN:=En, Data:=Data, FunctionType:=FunctionType,FunctionNumber:=FunctionNumber, ParameterDW:=ParameterDW, ParameterB:=ParameterB);

Done:=fbRPC.Done;
Executing:=fbRPC.Executing;
Waiting:=fbRPC.Waiting;
Error:=fbRPC.Error OR (fbRPC.Done AND fbRPC.ReturnValue<0);
Progress:=fbRPC.Progress;

END_FUNCTION_BLOCK

// ---- ComLib/POUs/Public/Level 1 Physical/ToAddress.TcPOU
{library PUBLIC}
(* Function to convert station number and device number to a valid address.
An address, is a number concatenated by SationNumber  and DeviceNumber and 
is defined as: StaionNumber*100+DeviceNumber, e.g., address 403 is Staion 4, Device 3.

NOTE: staion number must be in the range 1-INSTANCE_MAX_NUMBER_OF_STATIONS
          and device number in the range 1-INSTANCE_MAX_NUMBER_OF_DEVICES.

On success a valid address is returned otherwise -1.
*)
FUNCTION ToAddress :	INT
VAR_INPUT
	StationNumber:		INT;
	DeviceNumber:		INT;
END_VAR
VAR
END_VAR

ToAddress:=-1;

IF DeviceNumber>0 AND DeviceNumber<=ComGVL.INSTANCE_MAX_NUMBER_OF_DEVICES THEN
	IF StationNumber>0 AND StationNumber<=ComGVL.INSTANCE_MAX_NUMBER_OF_STATIONS THEN
		ToAddress:=StationNumber*100+DeviceNumber;
	END_IF;
END_IF;

END_FUNCTION

// ---- ComLib/POUs/Public/Level 6 Presentation/GetStatus.TcPOU
{library PUBLIC}
(* Function to get  current status of a device.
    This function can run continiously and will not block other communications.
    The validity/existence of the output values depends on the target device.   

    Note: that all outputs will always show a value but if hear beat is not continuously changing its an indication of dead communication.
    Frequency of the heart beat depends on communication speed and device execution speed.
 *)
FUNCTION_BLOCK GetStatus
VAR_INPUT
	En: 					BOOL:=FALSE;			(* Set to true to ask for status, the block  will continuously ask for status while true *)
END_VAR
VAR_OUTPUT
	Running:				BOOL:=FALSE;			(* True if the system is in running mode *)
	Progress:				INT:=0;					(* Progress (0-100) for last RPC call *)
	ProgramNumber:			INT:=0;					(* Program number for last RPC call *)
	HeartBeat:				BOOL:=FALSE;			(* On an active communication this signal will continuously change value *)
	Error: 					BOOL := FALSE;			(* True if an error occurred *)
END_VAR
VAR_IN_OUT
	Data: 					CommunicationData;		(* Common data structure to connect this function block to a specific Communicator block *)
END_VAR
VAR
	FunctionType: 			FUNCTION_TYPE;
	FunctionNumber: 		BYTE;
	ParameterDW:		DWORD;
	ParameterB:			BYTE;

	Done: 					BOOL:=FALSE;			(* If true, the command is transmitted ok, to reset set En to false *)
	Executing:				BOOL:=FALSE;			(* True while the command in transmitted *)
	Waiting:				BOOL:=FALSE;			(* True if the command is queued to be transmitted *)
	ReStart:				BOOL:=FALSE;

	fbRPC:					RPC1;
END_VAR

FunctionType:=FUNCTION_TYPE.FUNCTION_TYPE_INFORMATION;
FunctionNumber:=INT_TO_BYTE(INFO_FUNCTION_NUMBER.INFO_FUNCTION_RPC_STATUS);
ParameterDW:=0;										(* No parameters *)
ParameterB:=0;

fbRPC(EN:=En AND NOT ReStart AND NOT Data._Error, Data:=Data, FunctionType1:=FunctionType,FunctionNumber1:=FunctionNumber, ParameterDW1:=ParameterDW, ParameterB1:=ParameterB);

Done:=fbRPC.Done;
Executing:=fbRPC.Executing;
Waiting:=fbRPC.Waiting;
Error:=fbRPC.Error;

IF Done AND NOT Error THEN
	Data._ASyncProgress:=DWORD_TO_INT(SHR(fbRPC.ReturnValue2, 24) AND 16#FF);
	Data._ASyncStatus.FunctionNumber:=DWORD_TO_INT(SHR(fbRPC.ReturnValue2, 16) AND 16#FF);
	Data._ASyncStatus.Extra:=DWORD_TO_INT(fbRPC.ReturnValue2 AND 16#FF);
	Data._ASyncStatusCounter:=Data._ASyncStatusCounter+1;

	ReStart:=TRUE;
ELSIF Error AND NOT ReStart THEN
	ReStart:=TRUE;
ELSIF ReStart THEN
	ReStart:=FALSE;
END_IF;

Progress:=Data._ASyncStatus.Progress;
ProgramNumber:=Data._ASyncStatus.FunctionNumber;
Running:=Data._ASyncStatus.Extra=1;
HeartBeat:=UDINT_TO_BOOL(Data._ASyncStatusCounter MOD 2);

(* We need to copy global error flag *)
Error:=Data._Error;

END_FUNCTION_BLOCK

// ---- ComLib/POUs/Public/Level 5 Session/RPC Remote Procedural Call/RPC1.TcPOU
{library PUBLIC}
(*
RPC1 will handle RPC calls with 1 parameter.
A session will be established to the specific equipment during the function call and when a return value exist (or error) the session is ended.
Note, if FunctionType1 is set to ASync, RPC will only start a function and not wait for the function to end.

It is possible to queue many calls by cascade coupled blocks in serie or parallel.
By using the Done output signal as input to En on another function blockit is possible to serialise calls.

*)
FUNCTION_BLOCK RPC1
VAR_INPUT
	En: 			BOOL:=FALSE;			(* Set to true to call a  RPC 1 parameter function *)
	FunctionType1:	FUNCTION_TYPE;			(* Function type ASYNC or SYNC *)
	FunctionNumber1:INT;					(* RPC function number *)
	ParameterDW1:	DWORD;					(* DWORD parameter value *)
	ParameterB1:	BYTE;					(* Byte parameter value *)
END_VAR
VAR_OUTPUT
	Done: 				BOOL:=FALSE;			(* If true, the command is transmitted ok, to reset set En to false *)
	Executing:			BOOL:=FALSE;			(* True while the command in transmitted *)
	Waiting:			BOOL:=FALSE;			(* True if the command is queued to be transmitted *)
	Error: 				BOOL := FALSE;			(* True if an communication error occured *)
	ReturnValue1:		FUNCTION_TYPE;			(* Return value *)
	ReturnValue2:		DWORD;					(* DWORD return value *)
	ReturnValue3:		BYTE;						(* BYTE return value *)
END_VAR
VAR_IN_OUT
	Data: 				CommunicationData;		(* Common data structure to connect this function block to a specific Communicator block *)
END_VAR
VAR
	fbSessionInit: 		SessionInit;
	fbSessionSend: 	SessionSend;
	fbSessionEnd: 	SessionEnd;
	Memory: 			BOOL := FALSE;
END_VAR

fbSessionInit(En:=En, Data:=Data);
fbSessionSend(En:=fbSessionInit.Done, SessionID:=fbSessionInit.SessionID, Data:=Data,
                             FunctionType:=INT_TO_BYTE(FunctionType1), FunctionNumber:=INT_TO_BYTE(FunctionNumber1), ParameterDW:=ParameterDW1, ParameterB:=ParameterB1);

fbSessionEnd(En:=fbSessionSend.Done, Data:=Data);

Done:=fbSessionSend.Done;
Executing:=fbSessionSend.Executing;
Waiting:=fbSessionSend.Waiting;
Error:=fbSessionSend.Error;

IF fbSessionSend.Done AND NOT Memory THEN
	Memory:=TRUE;
	ReturnValue1:= fbSessionSend.Answer.FunctionType;  //BYTE_TO_FUNCTION_TYPE
	ReturnValue2:=fbSessionSend.Answer.ParameterDW;
	ReturnValue3:=fbSessionSend.Answer.ParameterB;
ELSIF NOT En THEN
	ReturnValue1:=FUNCTION_TYPE.FUNCTION_TYPE_ERROR_NO_FUNCTION;
	Memory:=FALSE;
ELSE
	Memory:=FALSE;
	ReturnValue1:=FUNCTION_TYPE.FUNCTION_TYPE_ERROR_BUSY;
END_IF;

END_FUNCTION_BLOCK

// ---- ComLib/POUs/Public/Level 6 Presentation/ABB/ABBGetStatus.TcPOU
{library PUBLIC}
(* Function to get robot status *)
FUNCTION_BLOCK ABBGetStatus
VAR_INPUT
	En: 					BOOL:=FALSE;			(* Set to true to ask for status *)
END_VAR
VAR_OUTPUT
	Done: 					BOOL:=FALSE;			(* If true, the command is transmitted ok, to reset set En to false *)
	Executing:				BOOL:=FALSE;			(* True while the command in transmitted *)
	Waiting:				BOOL:=FALSE;			(* True if the command is queued to be transmitted *)
	Error: 					BOOL := FALSE;			(* True if an error occured *)
	Progress:				INT:=0;							(* Return value *)
	RunningMode:			ABB_STATUS_RUNNING_MODE:=0;		(* Return value *)
	OperatingMode:			ABB_STATUS_OPERATING_MODE:=0;	(* Return value *)
	Running:				BOOL:=FALSE;					(* Return value *)
END_VAR
VAR_IN_OUT
	Data: 					CommunicationData;		(* Common data structure to connect this function block to a specific Communicator block *)
END_VAR
VAR
	FunctionType: 			FUNCTION_TYPE;
	FunctionNumber: 		BYTE;
	ParameterDW:			DWORD;
	ParameterB:				BYTE;
	Sequence:				INT:=0;

	fbRPC:					RPC1;
END_VAR


FunctionType:=FUNCTION_TYPE.FUNCTION_TYPE_INFORMATION;
FunctionNumber:=INT_TO_BYTE(INFO_FUNCTION_NUMBER.INFO_FUNCTION_SYSTEM_STATUS);
ParameterDW:=0;										(* No parameters *)
ParameterB:=0;

fbRPC(EN:=En, Data:=Data, FunctionType1:=FunctionType,FunctionNumber1:=FunctionNumber, ParameterDW1:=ParameterDW, ParameterB1:=ParameterB);

Done:=fbRPC.Done;
Executing:=fbRPC.Executing;
Waiting:=fbRPC.Waiting;
Error:=fbRPC.Error;

Progress:=DWORD_TO_INT(SHR(fbRPC.ReturnValue2, 24) AND 16#FF);
RunningMode:=DWORD_TO_INT(SHR(fbRPC.ReturnValue2, 16) AND 16#FF);  
OperatingMode:=DWORD_TO_INT(SHR(fbRPC.ReturnValue2, 8) AND 16#FF); 
Running:=DWORD_TO_BOOL(fbRPC.ReturnValue2 AND 16#FF);

END_FUNCTION_BLOCK

// ---- ComLib/POUs/Public/Level 6 Presentation/ABB/Goto/ABBGoToSensor.TcPOU
{library PUBLIC}
(* Function to send a robot to sensor location *)
FUNCTION_BLOCK ABBGoToSensor
VAR_INPUT
	En: 				BOOL:=FALSE;				(* Set to true to start *)
END_VAR
VAR_OUTPUT
	Done: 				BOOL:=FALSE;			(* If true, the command is transmitted ok, to reset set En to false *)
	Executing:			BOOL:=FALSE;			(* True while the command in transmitted *)
	Waiting:			BOOL:=FALSE;			(* True if the command is queued to be transmitted *)
	Error: 				BOOL := FALSE;			(* True if an error occured *)
	Progress:			INT:=0;						(* Function progress *)
END_VAR
VAR_IN_OUT
	Data: 				CommunicationData;		(* Common data structure to connect this function block to a specific Communicator block *)
END_VAR
VAR
	FunctionType: 		FUNCTION_TYPE;
	FunctionNumber: 	INT;
	ParameterDW:		DWORD;
	ParameterB:			BYTE;
	Sequence:			INT:=0;

	fbRPC:				ASyncRPC;
END_VAR

FunctionType:=FUNCTION_TYPE.FUNCTION_TYPE_ASYNC_RPC;
FunctionNumber:=ABB_ASYNC_FUNCTION_GOTO_SENSOR;
ParameterDW:=0;										(* No parameters *)
ParameterB:=0;

fbRPC(EN:=En, Data:=Data, FunctionType:=FunctionType,FunctionNumber:=FunctionNumber, ParameterDW:=ParameterDW, ParameterB:=ParameterB);

Done:=fbRPC.Done;
Executing:=fbRPC.Executing;
Waiting:=fbRPC.Waiting;
Error:=fbRPC.Error OR (fbRPC.Done AND fbRPC.ReturnValue<0);
Progress:=fbRPC.Progress;

END_FUNCTION_BLOCK

// ---- ComLib/POUs/Public/Level 6 Presentation/ABB/Goto/ABBGoToStorage.TcPOU
{library PUBLIC}
(* Function to send a robot to storage location *)
FUNCTION_BLOCK ABBGoToStorage
VAR_INPUT
	En: 			BOOL:=FALSE;			(* Set to true to start *)
END_VAR
VAR_OUTPUT
	Done: 			BOOL:=FALSE;			(* If true, the command is transmitted ok, to reset set En to false *)
	Executing:		BOOL:=FALSE;			(* True while the command in transmitted *)
	Waiting:		BOOL:=FALSE;			(* True if the command is queued to be transmitted *)
	Error: 			BOOL:= FALSE;			(* True if an error occured *)
	Progress:		INT:=0;					(* Function progress *)
END_VAR
VAR_IN_OUT
	Data: 			CommunicationData;		(* Common data structure to connect this function block to a specific Communicator block *)
END_VAR
VAR
	FunctionType: 	FUNCTION_TYPE;
	FunctionNumber: INT;
	ParameterDW:	DWORD;
	ParameterB:		BYTE;
	Sequence:		INT:=0;

	fbRPC:			ASyncRPC;
END_VAR


FunctionType:=FUNCTION_TYPE.FUNCTION_TYPE_ASYNC_RPC;
FunctionNumber:=ABB_ASYNC_FUNCTION_GOTO_STORAGE;
ParameterDW:=0;										(* No parameters *)
ParameterB:=0;

fbRPC(EN:=En, Data:=Data, FunctionType:=FunctionType,FunctionNumber:=FunctionNumber, ParameterDW:=ParameterDW, ParameterB:=ParameterB);

Done:=fbRPC.Done;
Executing:=fbRPC.Executing;
Waiting:=fbRPC.Waiting;
Error:=fbRPC.Error OR (fbRPC.Done AND fbRPC.ReturnValue<0);
Progress:=fbRPC.Progress;

END_FUNCTION_BLOCK

// ---- ComLib/POUs/Public/Level 6 Presentation/ABB/Goto/ABBGoToConveyor1.TcPOU
{library PUBLIC}
(* Function to send a robot to storage location *)
FUNCTION_BLOCK ABBGoToConveyor1
VAR_INPUT
	En: 			BOOL:=FALSE;				(* Set to true to start *)
END_VAR
VAR_OUTPUT
	Done: 				BOOL:=FALSE;			(* If true, the command is transmitted ok, to reset set En to false *)
	Executing:			BOOL:=FALSE;			(* True while the command in transmitted *)
	Waiting:			BOOL:=FALSE;			(* True if the command is queued to be transmitted *)
	Error: 				BOOL := FALSE;			(* True if an error occured *)
	Progress:			INT:=0;					(* Function progress *)
END_VAR
VAR_IN_OUT
	Data: 				CommunicationData;		(* Common data structure to connect this function block to a specific Communicator block *)
END_VAR
VAR
	FunctionType: 		FUNCTION_TYPE;
	FunctionNumber: 	INT;
	ParameterDW:	DWORD;
	ParameterB:		BYTE;
	Sequence:			INT:=0;

	fbRPC:				ASyncRPC;
END_VAR

FunctionType:=FUNCTION_TYPE.FUNCTION_TYPE_ASYNC_RPC;
FunctionNumber:=ABB_ASYNC_FUNCTION_GOTO_CONVEYOR_1;
ParameterDW:=0;										(* No parameters *)
ParameterB:=0;

fbRPC(EN:=En, Data:=Data, FunctionType:=FunctionType,FunctionNumber:=FunctionNumber, ParameterDW:=ParameterDW, ParameterB:=ParameterB);

Done:=fbRPC.Done;
Executing:=fbRPC.Executing;
Waiting:=fbRPC.Waiting;
Error:=fbRPC.Error OR (fbRPC.Done AND fbRPC.ReturnValue<0);
Progress:=fbRPC.Progress;

END_FUNCTION_BLOCK

// ---- ComLib/POUs/Public/Level 6 Presentation/ABB/Goto/ABBGoToConveyor2.TcPOU
{library PUBLIC}
(* Function to send a robot to storage location *)
FUNCTION_BLOCK ABBGoToConveyor2
VAR_INPUT
	En: 			BOOL:=FALSE;				(* Set to true to start *)
END_VAR
VAR_OUTPUT
	Done: 				BOOL:=FALSE;			(* If true, the command is transmitted ok, to reset set En to false *)
	Executing:			BOOL:=FALSE;			(* True while the command in transmitted *)
	Waiting:			BOOL:=FALSE;			(* True if the command is queued to be transmitted *)
	Error: 				BOOL := FALSE;			(* True if an error occured *)
	Progress:			INT:=0;						(* Function progress *)
END_VAR
VAR_IN_OUT
	Data: 				CommunicationData;		(* Common data structure to connect this function block to a specific Communicator block *)
END_VAR
VAR
	FunctionType: 		FUNCTION_TYPE;
	FunctionNumber: 	INT;
	ParameterDW:	DWORD;
	ParameterB:		BYTE;
	Sequence:			INT:=0;

	fbRPC:				ASyncRPC;
END_VAR

FunctionType:=FUNCTION_TYPE.FUNCTION_TYPE_ASYNC_RPC;
FunctionNumber:=ABB_ASYNC_FUNCTION_GOTO_CONVEYOR_2;
ParameterDW:=0;										(* No parameters *)
ParameterB:=0;

fbRPC(EN:=En, Data:=Data, FunctionType:=FunctionType,FunctionNumber:=FunctionNumber, ParameterDW:=ParameterDW, ParameterB:=ParameterB);

Done:=fbRPC.Done;
Executing:=fbRPC.Executing;
Waiting:=fbRPC.Waiting;
Error:=fbRPC.Error OR (fbRPC.Done AND fbRPC.ReturnValue<0);
Progress:=fbRPC.Progress;

END_FUNCTION_BLOCK

// ---- ComLib/POUs/Public/Level 6 Presentation/ABB/Pick Leave/ABBPickLeaveSensor.TcPOU
{library PUBLIC}
(* Function to start a pick or leave operation *)
FUNCTION_BLOCK ABBPickLeaveSensor
VAR_INPUT
	En: 			BOOL:=FALSE;				(* Set to true to start *)
	Pick:			BOOL:=TRUE;					(* If true pick operation, if false leave operation *)
	Position:		INT:=0;						(* Position number not used *)
END_VAR
VAR_OUTPUT
	Done: 				BOOL:=FALSE;			(* If true, the command is transmitted ok, to reset set En to false *)
	Executing:			BOOL:=FALSE;			(* True while the command in transmitted *)
	Waiting:			BOOL:=FALSE;			(* True if the command is queued to be transmitted *)
	Error: 				BOOL := FALSE;			(* True if an error occured *)
	Progress:			INT:=0;					(* Function progress *)
END_VAR
VAR_IN_OUT
	Data: 				CommunicationData;		(* Common data structure to connect this function block to a specific Communicator block *)
END_VAR
VAR
	FunctionType: 		FUNCTION_TYPE;
	FunctionNumber: 	INT;
	ParameterDW:	DWORD;
	ParameterB:		BYTE;
	Sequence:			INT:=0;

	fbRPC:				ASyncRPC;
END_VAR


FunctionType:=FUNCTION_TYPE.FUNCTION_TYPE_ASYNC_RPC;
FunctionNumber:=ABB_ASYNC_FUNCTION_PL_SENSOR;
ParameterDW:=INT_TO_DWORD(Position);
ParameterB:=BOOL_TO_BYTE(Pick);

fbRPC(EN:=En, Data:=Data, FunctionType:=FunctionType,FunctionNumber:=FunctionNumber, ParameterDW:=ParameterDW, ParameterB:=ParameterB);

Done:=fbRPC.Done;
Executing:=fbRPC.Executing;
Waiting:=fbRPC.Waiting;
Error:=fbRPC.Error OR (fbRPC.Done AND fbRPC.ReturnValue<0);
Progress:=fbRPC.Progress;

END_FUNCTION_BLOCK

// ---- ComLib/POUs/Public/Level 6 Presentation/ABB/Pick Leave/ABBPickLeaveStorage.TcPOU
{library PUBLIC}
(* Function to start a pick or leave operation *)
FUNCTION_BLOCK ABBPickLeaveStorage
VAR_INPUT
	En: 				BOOL:=FALSE;			(* Set to true to start *)
	Pick:				BOOL:=TRUE;				(* If true pick operation, if false leave operation *)
	Position:			INT:=0;					(* Position number 1-9 *)
END_VAR
VAR_OUTPUT
	Done: 				BOOL:=FALSE;			(* If true, the command is transmitted ok, to reset set En to false *)
	Executing:			BOOL:=FALSE;			(* True while the command in transmitted *)
	Waiting:			BOOL:=FALSE;			(* True if the command is queued to be transmitted *)
	Error: 				BOOL := FALSE;			(* True if an error occured *)
	Progress:			INT:=0;					(* Function progress *)
END_VAR
VAR_IN_OUT
	Data: 				CommunicationData;		(* Common data structure to connect this function block to a specific Communicator block *)
END_VAR
VAR
	FunctionType: 		FUNCTION_TYPE;
	FunctionNumber: 	INT;
	ParameterDW:		DWORD;
	ParameterB:			BYTE;
	Sequence:			INT:=0;

	fbRPC:				ASyncRPC;
END_VAR


FunctionType:=FUNCTION_TYPE.FUNCTION_TYPE_ASYNC_RPC;
FunctionNumber:=ABB_ASYNC_FUNCTION_PL_STORAGE;
ParameterDW:=INT_TO_DWORD(Position);
ParameterB:=BOOL_TO_BYTE(Pick);

fbRPC(EN:=En, Data:=Data, FunctionType:=FunctionType,FunctionNumber:=FunctionNumber, ParameterDW:=ParameterDW, ParameterB:=ParameterB);

Done:=fbRPC.Done;
Executing:=fbRPC.Executing;
Waiting:=fbRPC.Waiting;
Error:=fbRPC.Error OR (fbRPC.Done AND fbRPC.ReturnValue<0);
Progress:=fbRPC.Progress;

END_FUNCTION_BLOCK

// ---- ComLib/POUs/Public/Level 6 Presentation/ABB/Pick Leave/ABBPickLeaveTable.TcPOU
{library PUBLIC}
(* Function to start a pick or leave operation *)
FUNCTION_BLOCK ABBPickLeaveTable
VAR_INPUT
	En: 				BOOL:=FALSE;			(* Set to true to start *)
	Pick:				BOOL:=TRUE;				(* If true pick operation, if false leave operation *)
	Position:			INT:=0;					(* Position number, 1=brick, 2=rod, 3=assembly *)
END_VAR
VAR_OUTPUT
	Done: 				BOOL:=FALSE;			(* If true, the command is transmitted ok, to reset set En to false *)
	Executing:			BOOL:=FALSE;			(* True while the command in transmitted *)
	Waiting:			BOOL:=FALSE;			(* True if the command is queued to be transmitted *)
	Error: 				BOOL := FALSE;			(* True if an error occured *)
	Progress:			INT:=0;					(* Function progress *)
END_VAR
VAR_IN_OUT
	Data: 				CommunicationData;		(* Common data structure to connect this function block to a specific Communicator block *)
END_VAR
VAR
	FunctionType: 		FUNCTION_TYPE;
	FunctionNumber: 	INT;
	ParameterDW:		DWORD;
	ParameterB:			BYTE;
	Sequence:			INT:=0;

	fbRPC:				ASyncRPC;
END_VAR


FunctionType:=FUNCTION_TYPE.FUNCTION_TYPE_ASYNC_RPC;
FunctionNumber:=ABB_ASYNC_FUNCTION_PL_TABLE;
ParameterDW:=INT_TO_DWORD(Position);
ParameterB:=BOOL_TO_BYTE(Pick);

fbRPC(EN:=En, Data:=Data, FunctionType:=FunctionType,FunctionNumber:=FunctionNumber, ParameterDW:=ParameterDW, ParameterB:=ParameterB);

Done:=fbRPC.Done;
Executing:=fbRPC.Executing;
Waiting:=fbRPC.Waiting;
Error:=fbRPC.Error OR (fbRPC.Done AND fbRPC.ReturnValue<0);
Progress:=fbRPC.Progress;

END_FUNCTION_BLOCK

// ---- ComLib/POUs/Public/Level 6 Presentation/ABB/Pick Leave/ABBPickLeaveConveyor1.TcPOU
{library PUBLIC}
(* Function to start a pick or leave operation *)
FUNCTION_BLOCK ABBPickLeaveConveyor1
VAR_INPUT
	En: 			BOOL:=FALSE;				(* Set to true to start *)
	Pick:			BOOL:=TRUE;					(* If true pick operation, if false leave operation *)
	Position:		INT:=0;						(* Position number not used *)
END_VAR
VAR_OUTPUT
	Done: 				BOOL:=FALSE;			(* If true, the command is transmitted ok, to reset set En to false *)
	Executing:			BOOL:=FALSE;			(* True while the command in transmitted *)
	Waiting:			BOOL:=FALSE;			(* True if the command is queued to be transmitted *)
	Error: 				BOOL := FALSE;			(* True if an error occured *)
	Progress:			INT:=0;					(* Function progress *)
END_VAR
VAR_IN_OUT
	Data: 				CommunicationData;		(* Common data structure to connect this function block to a specific Communicator block *)
END_VAR
VAR
	FunctionType: 		FUNCTION_TYPE;
	FunctionNumber: 	INT;
	ParameterDW:		DWORD;
	ParameterB:			BYTE;
	Sequence:			INT:=0;

	fbRPC:				ASyncRPC;
END_VAR


FunctionType:=FUNCTION_TYPE.FUNCTION_TYPE_ASYNC_RPC;
FunctionNumber:=ABB_ASYNC_FUNCTION_PL_CONVEYOR_1;
ParameterDW:=INT_TO_DWORD(Position);
ParameterB:=BOOL_TO_BYTE(Pick);

fbRPC(EN:=En, Data:=Data, FunctionType:=FunctionType,FunctionNumber:=FunctionNumber, ParameterDW:=ParameterDW, ParameterB:=ParameterB);

Done:=fbRPC.Done;
Executing:=fbRPC.Executing;
Waiting:=fbRPC.Waiting;
Error:=fbRPC.Error OR (fbRPC.Done AND fbRPC.ReturnValue<0);
Progress:=fbRPC.Progress;

END_FUNCTION_BLOCK

// ---- ComLib/POUs/Public/Level 6 Presentation/ABB/Pick Leave/ABBPickLeaveConveyor2.TcPOU
{library PUBLIC}
(* Function to start a pick or leave operation *)
FUNCTION_BLOCK ABBPickLeaveConveyor2
VAR_INPUT
	En: 			BOOL:=FALSE;				(* Set to true to start *)
	Pick:			BOOL:=TRUE;					(* If true pick operation, if false leave operation *)
	Position:		INT:=0;						(* Position number not used *)
END_VAR
VAR_OUTPUT
	Done: 				BOOL:=FALSE;			(* If true, the command is transmitted ok, to reset set En to false *)
	Executing:			BOOL:=FALSE;			(* True while the command in transmitted *)
	Waiting:			BOOL:=FALSE;			(* True if the command is queued to be transmitted *)
	Error: 				BOOL := FALSE;			(* True if an error occured *)
	Progress:			INT:=0;					(* Function progress *)
END_VAR
VAR_IN_OUT
	Data: 				CommunicationData;		(* Common data structure to connect this function block to a specific Communicator block *)
END_VAR
VAR
	FunctionType: 		FUNCTION_TYPE;
	FunctionNumber: 	INT;
	ParameterDW:		DWORD;
	ParameterB:			BYTE;
	Sequence:			INT:=0;

	fbRPC:				ASyncRPC;
END_VAR


FunctionType:=FUNCTION_TYPE.FUNCTION_TYPE_ASYNC_RPC;
FunctionNumber:=ABB_ASYNC_FUNCTION_PL_CONVEYOR_2;
ParameterDW:=INT_TO_DWORD(Position);
ParameterB:=BOOL_TO_BYTE(Pick);

fbRPC(EN:=En, Data:=Data, FunctionType:=FunctionType,FunctionNumber:=FunctionNumber, ParameterDW:=ParameterDW, ParameterB:=ParameterB);

Done:=fbRPC.Done;
Executing:=fbRPC.Executing;
Waiting:=fbRPC.Waiting;
Error:=fbRPC.Error OR (fbRPC.Done AND fbRPC.ReturnValue<0);
Progress:=fbRPC.Progress;

END_FUNCTION_BLOCK

// ---- ComLib/POUs/Public/Level 6 Presentation/Gantry/GantryPick.TcPOU
{library PUBLIC}
(* Function to pick a pallet from a specific station and position. *)
FUNCTION_BLOCK GantryPick
VAR_INPUT
	En: 				BOOL:=FALSE;			(* Set to true to start *)
	PickStation:		StationType;			(* Station number 1-4 to pick from *)
	PickPosition:		PositionType;			(* Position number 1-9 to pick from *)
END_VAR
VAR_OUTPUT
	Done: 				BOOL:=FALSE;			(* If true, the command is transmitted ok, to reset set En to false *)
	Executing:			BOOL:=FALSE;			(* True while the command in transmitted *)
	Waiting:			BOOL:=FALSE;			(* True if the command is queued to be transmitted *)
	Error: 				BOOL := FALSE;			(* True if an error occured *)
	Progress:			INT:=0;					(* Function progress *)
END_VAR
VAR_IN_OUT
	Data: 				CommunicationData;		(* Common data structure to connect this function block to a specific Communicator block *)
END_VAR
VAR
	FunctionType: 		FUNCTION_TYPE;
	FunctionNumber: 	INT;
	ParameterDW:	DWORD;
	ParameterB:		BYTE;
	ParametersOK:	BOOL;

	fbRPC:				ASyncRPC;
END_VAR


